            // ---- Engineering → % scaling ----
            IF enableScaling THEN
                pvPct := _ScaleToPct(pvEngFiltered,       pLoEng, pHiEng);
                spPct := _ScaleToPct(processSetpointAuto, pLoEng, pHiEng);
            ELSE
                pvPct := pvEngFiltered;        // already %
                spPct := processSetpointAuto;  // already %
            END_IF

            // ---- Manual path (HMI) ----
            manualCmd := LIMIT(0.0, processSetpointMan, 100.0);

            // Reverse/direct action by Kp sign
            IF reverseActing THEN
                kpUse := -ABS(kp);
            ELSE
                kpUse :=  ABS(kp);
            END_IF

            // ===================== PV HOLD behavior =====================
            // When PV hold active: keep motor energized, force reference=0.0,
            // and hold PID (avoid error/windup) by forcing SET=ACT and MAN=TRUE.
            IF pvHoldActive THEN

                deviceState := 'Running (PV hold: output inhibited)';
                vfdStartCmdOut := TRUE;        // keep energized
                running := TRUE;               // keep permissives (change to FALSE if you prefer)

                instPID(
                    ACT := pvPct,
                    SET := pvPct,              // hold: SET follows PV -> DIFF ~ 0
                    M_I := 0.0,                // forced output during hold
                    MAN := TRUE,               // hold PID
                    RST := resetPID,
                    KP  := kpUse,
                    TN  := tn,
                    TV  := tv,
                    LL  := outLowLimitPct,
                    LH  := outHighLimitPct,
                    Y   => yPID,
                    DIFF=> pidDiff,
                    LIM => pidLimited
                );

                // Output inhibited to zero, motor stays enabled
                controlOutputPct := 0.0;

            ELSE
                // ===================== Normal control =====================
                instPID(
                    ACT := pvPct,
                    SET := spPct,
                    M_I := manualCmd,
                    MAN := NOT autoMode,
                    RST := resetPID,
                    KP  := kpUse,
                    TN  := tn,
                    TV  := tv,
                    LL  := outLowLimitPct,
                    LH  := outHighLimitPct,
                    Y   => yPID,
                    DIFF=> pidDiff,
                    LIM => pidLimited
                );

                // Mode select, offset, clamp
                IF autoMode THEN
                    controlOutputPct := yPID;
                ELSE
                    controlOutputPct := manualCmd;
                END_IF

                controlOutputPct := LIMIT(outLowLimitPct, controlOutputPct + outputOffsetPct, outHighLimitPct);
            END_IF
        END_IF

    // ------------------------------------------------------------
    90: // Stopping (normal, de-energize)
        running := FALSE;
        controlOutputPct := 0.0;
        vfdStartCmdOut := FALSE;
        tonRunFbWait(IN := FALSE);

        // Return to Idle once stop released and safety OK
        IF NOT stopCommand AND allSafetyOK THEN
            deviceState := 'Idle';
            step := 0;
        END_IF

    // ------------------------------------------------------------
    ELSE
        running := FALSE;
        controlOutputPct := 0.0;
        deviceState := 'Idle';
        vfdStartCmdOut := FALSE;
        step := 0;
END_CASE;


// =============================== Status code ===============================
IF vfdFaultFeedback THEN
    statusCode := 2;             // Fault
ELSIF running THEN
    statusCode := 1;             // Running
ELSE
    statusCode := 0;             // Idle
END_IF

// HMI feedbacks & status (encapsulates PT1 displays and status code if desired)
_FeedbackDisplay();

// Setpoint input handling (encapsulates TUNE2-based HMI writes & nudges)
_SetpointInputControl();

METHOD _FeedbackDisplay
VAR_INPUT
END_VAR
//instPT1_WhiteWaterSiloDisplay
//whiteWaterLevelDisplay
// 5) HMI DISPLAY SIGNALS (filtered speeds/torques + GROUP status)
instPT1_SpeedDisplay(in := vfdEngFeedback, T := displayFilterTime, K := 1.0, out => vfdEngDisplay);
instPT1_TorqueDisplay (in := vfdTorqueFeedback , T := displayFilterTime, K := 1.0, out => vfdTorqueDisplay);
instPT1_ProcessFeedbackEngDisplay(in := wirePitLevel , T := displayFilterTime, K := 1.0, out => wirePitLevelDisplay);
instPT1_WhiteWaterSiloLevelDisplay(in := whiteWaterSiloLevel , T := displayFilterTime, K := 1.0, out => whiteWaterSiloLevelDisplay);
END_METHOD

// ============================ Helper ============================
METHOD PRIVATE _ScaleToPct : REAL
VAR_INPUT
    xEng  : REAL;  // value in engineering units
    loEng : REAL;  // min eng
    hiEng : REAL;  // max eng
END_VAR
VAR
    span : REAL;
    pct  : REAL;
END_VAR

span := hiEng - loEng;
IF span = 0.0 THEN
    _ScaleToPct := 0.0; // avoid div by zero
ELSE
    pct := (xEng - loEng) / span * 100.0;
    _ScaleToPct := LIMIT(0.0, pct, 100.0);
END_IF
END_METHOD

// ============================================================================
// METHOD: _SetpointInputControl
// Purpose: Handle HMI writes for manual output using OSCAT TUNE2. Any external
//          write to manualOutputPct bigger than the configured step will pulse
//          SET for one scan. No SU/SD buttons here (PressureCtrl doesn’t use them).
// Objetivo: Tratar escrita da HMI no manualOutputPct via TUNE2. Mudança externa
//           > passo gera pulso SET de 1 varredura. Sem botões ↑/↓ neste FB.
// ============================================================================
METHOD PRIVATE _SetpointInputControl
VAR
    spManClamped : REAL;
    spAutoClamped : REAL;
	
END_VAR
// Detect external write (> step): ignore tiny jitter
IF ABS(processSetpointMan - processSetpointManOld) > instTUNE2ManSetpoint.SS THEN
    // Clamp to output limits before writing (garante limites)
    spManClamped := LIMIT(outLowLimitPct, processSetpointMan, outHighLimitPct);

    // One-scan SET pulse into TUNE2 (pulso SET de 1 ciclo)
    instTUNE2ManSetpoint(
        SET_val := spManClamped,
        SET     := TRUE
    );
    instTUNE2ManSetpoint(SET := FALSE);

    // Remember applied value (memoriza)
    processSetpointManOld := processSetpointMan;
ELSE
    // Track last seen to avoid drift (rastreia último observado)
    processSetpointManOld := processSetpointMan;
END_IF;

// Keep TUNE2 active (no SU/SD in this FB)
instTUNE2ManSetpoint(
    SET      := FALSE,
    SU       := processSetpointManInc,
    SD       := processSetpointManDec,
    RST      := FALSE,
    SS       := 0.1,           // step reference (passo de referência)
    FS       := 0.0,                     // unused
    LIMIT_L  := outLowLimitPct,
    LIMIT_H  := outHighLimitPct,
    Y        => processSetpointMan
);




// Detect external write (> step): ignore tiny jitter
IF ABS(processSetpointAuto - processSetpointAutoOld) > instTUNE2AutoSetpoint.SS THEN
    // Clamp to output limits before writing (garante limites)
    spAutoClamped := LIMIT(0, processSetpointAuto, 100);

    // One-scan SET pulse into TUNE2 (pulso SET de 1 ciclo)
    instTUNE2AutoSetpoint(
        SET_val := spAutoClamped,
        SET     := TRUE
    );
    instTUNE2AutoSetpoint(SET := FALSE);

    // Remember applied value (memoriza)
    processSetpointAutoOld := processSetpointAuto;
ELSE
    // Track last seen to avoid drift (rastreia último observado)
    processSetpointAutoOld := processSetpointAuto;
END_IF;

// Keep TUNE2 active (no SU/SD in this FB)
instTUNE2AutoSetpoint(
    SET      := FALSE,
    SU       := processSetpointAutoInc,
    SD       := processSetpointAutoDec,
    RST      := FALSE,
    SS       := 0.1,           // step reference (passo de referência)
    FS       := 0.0,                     // unused
    LIMIT_L  := 0.0,
    LIMIT_H  := 100.0,
    Y        => processSetpointAuto
);
END_METHOD

END_FUNCTION_BLOCK

// ---- Function Blocks/PaperMachine/Auxiliary/FB_StockPumpFlowControl.TcPOU
(*
    FB_StockPumpFlowControl

    Purpose:
    Dedicated dry-stock flow controller for the Stock Pump (P1_100_UG05).
    The existing Mix Pump (P1_100_UG01) is the approach-flow fan/mix pump and
    is intentionally outside the scope of this function block.

    First delivery:
    Public interface and method declarations only. No control logic is active.
*)

FUNCTION_BLOCK FB_StockPumpFlowControl
VAR_INPUT
    // ===== General enable and sequence commands =====
    enable                              : BOOL;
    processPermissive                   : BOOL;
    startCommand                        : BOOL;
    stopCommand                         : BOOL;
    resetCommand                        : BOOL;
    autoMode                            : BOOL;   // TRUE=Automatic / FALSE=Manual
    machineRunning                      : BOOL;
    processStable                       : BOOL;

    // ===== Manual speed-reference adjustment =====
    stockPumpSetpointManInc             : BOOL;   // Increase manual speed reference
    stockPumpSetpointManDec             : BOOL;   // Decrease manual speed reference
    manualSetpointStepPct               : REAL := 0.1;

    // ===== Process inputs =====
    basisWeightSetpointGm2              : REAL;   // Desired basis weight [g/m2]
    effectiveWidthM                     : REAL;   // Effective sheet/jet width [m]
    wireSpeedMPM                        : REAL;   // Forming wire speed [m/min]
    stockConsistencyPct                 : REAL;   // Stock consistency [%], e.g. 3.5 = 3.5%
    stockConsistencySignalValid         : BOOL;
    refinedStockTankConsistencyPct      : REAL;   // Refined-stock tank consistency indication [%]
    refinedStockTankConsistencySignalValid : BOOL;
    stockFlowFeedbackM3h                : REAL;   // Measured suspension flow [m3/h]
    stockFlowSignalValid                : BOOL;
    stockTankLevelPct                   : REAL;   // Stock-tank level, already scaled [%]
    stockTankLevelSignalValid           : BOOL;

    // ===== Production correction factors =====
    recipeCalibrationFactor             : REAL := 1.0;
    operatorTrimFactor                  : REAL := 1.0;
    basisWeightLabGm2                   : REAL;
    calculateCalibrationCommand         : BOOL;

    // ===== PID parameters =====
    kp                                  : REAL := 1.0;
    tn                                  : REAL := 8.0;     // Integral time [s]
    tv                                  : REAL := 0.0;     // Derivative time [s]
    pidDeadbandM3h                      : REAL := 0.0;     // Flow deadband [m3/h]
    resetPID                            : BOOL;

    // ===== Process engineering limits =====
    stockDensityKgM3                    : REAL := 1000.0;
    minimumValidConsistencyPct          : REAL := 0.1;
    maximumValidConsistencyPct          : REAL := 10.0;
    minimumStockFlowM3h                 : REAL := 0.0;
    maximumStockFlowM3h                 : REAL := 250.0;
    standbyStockFlowM3h                 : REAL := 0.0;
    minimumAutomaticWireSpeedMPM        : REAL := 0.0;

    // ===== Calibration and trim limits =====
    minimumRecipeCalibrationFactor      : REAL := 0.5;
    maximumRecipeCalibrationFactor      : REAL := 1.5;
    minimumOperatorTrimFactor           : REAL := 0.95;
    maximumOperatorTrimFactor           : REAL := 1.05;

    // ===== Filters and ramps =====
    consistencyFilterTime               : TIME := T#5s;
    flowFeedbackFilterTime              : TIME := T#1s;
    stockTankLevelFilterTime            : TIME := T#2s;
    stockFlowSetpointRampUpM3hS         : REAL := 1.0;
    stockFlowSetpointRampDownM3hS       : REAL := 1.0;
    speedReferenceRampUpPctS            : REAL := 10.0;
    speedReferenceRampDownPctS          : REAL := 10.0;

    // ===== Speed-reference limits =====
    minimumSpeedReferencePct            : REAL := 0.0;
    maximumSpeedReferencePct            : REAL := 100.0;

    // ===== Signal fallback and alarm timing =====
    invalidConsistencyGraceTime         : TIME := T#5s;
    automaticStabilizationTime          : TIME := T#10s;
    flowDeviationWarningPct             : REAL := 5.0;
    flowDeviationAlarmPct               : REAL := 10.0;
    flowDeviationWarningDelay           : TIME := T#10s;
    flowDeviationAlarmDelay             : TIME := T#20s;

    // ===== Drive interface and supervision =====
    vfdReady                            : BOOL;
    vfdRunFeedback                      : BOOL;
    vfdFaultFeedback                    : BOOL;
    vfdRunFbTimeout                     : TIME := T#5s;
    vfdCurrentFeedback                  : REAL;
    vfdSpeedFeedbackPct                 : REAL;
    vfdTorqueFeedback                   : REAL;

    // ===== Safety and process interlocks =====
    safetyOk                            : BOOL := TRUE;
    estopOk                             : BOOL := TRUE;
    guardClosedOk                       : BOOL := TRUE;
    interlock1                          : BOOL := TRUE;
    interlock2                          : BOOL := TRUE;
    interlock3                          : BOOL := TRUE;
    interlock4                          : BOOL := TRUE;
    interlock5                          : BOOL := TRUE;
    interlock6                          : BOOL := TRUE;
END_VAR

VAR_IN_OUT
    // Existing HMI manual reference can be connected here without duplicating it.
    manualSpeedSetpointPct              : REAL;
END_VAR

VAR_OUTPUT
    // ===== Drive commands =====
    vfdStartCmdOut                      : BOOL;
    vfdResetCmdOut                      : BOOL;
    speedReferencePct                   : REAL;

    // ===== Flow and dry-mass calculation =====
    dryMassSetpointKgH                  : REAL;
    dryMassFeedbackKgH                  : REAL;
    stockFlowTheoreticalM3h             : REAL;
    stockFlowCorrectedM3h               : REAL;
    stockFlowLimitedM3h                 : REAL;
    stockFlowSetpointM3h                : REAL;
    stockFlowFeedbackFilteredM3h        : REAL;
    stockConsistencyFilteredPct         : REAL;
    stockConsistencyUsedPct             : REAL;

    // ===== Refined-stock tank consistency indication =====
    refinedStockTankConsistencyFilteredPct : REAL;
    refinedStockTankConsistencySignalInvalid : BOOL;

    // ===== Stock-tank indication =====
    stockTankLevelFilteredPct           : REAL;
    stockTankLevelSignalInvalid         : BOOL;

    // ===== PID diagnostics =====
    pidErrorM3h                         : REAL;
    pidOutputPct                        : REAL;
    pidOutputSaturated                  : BOOL;

    // ===== Calibration diagnostics =====
    suggestedCalibrationFactor         : REAL;
    suggestedCalibrationFactorValid    : BOOL;

    // ===== Validation and limitation status =====
    flowCalculationValid                : BOOL;
    automaticControlValid               : BOOL;
    automaticControlInvalid             : BOOL;
    consistencySignalInvalid            : BOOL;
    flowSignalInvalid                   : BOOL;
    basisWeightSetpointInvalid          : BOOL;
    effectiveWidthInvalid               : BOOL;
    wireSpeedInvalid                    : BOOL;
    calibrationFactorInvalid            : BOOL;
    operatorTrimFactorInvalid           : BOOL;
    flowSetpointLimited                 : BOOL;
    speedReferenceLimited              : BOOL;
    calculationUsingLastValidConsistency : BOOL;

    // ===== Deviation alarms =====
    flowDeviationWarning                : BOOL;
    flowDeviationAlarm                  : BOOL;
    warningActive                       : BOOL;
    alarmActive                         : BOOL;

    // ===== Operating state =====
    running                             : BOOL;
    controlActive                       : BOOL;
    manualActive                        : BOOL;
    automaticActive                     : BOOL;
    statusCode                          : INT;
    deviceState                         : STRING(80);

    // ===== Drive feedback displays =====
    vfdCurrentDisplay                   : REAL;
    vfdSpeedDisplayPct                  : REAL;
    vfdTorqueDisplay                    : REAL;
END_VAR

VAR
    // ===== Initialization and command edges =====
    firstScan                           : BOOL := TRUE;
    startCommandOld                     : BOOL;
    stopCommandOld                      : BOOL;
    resetCommandOld                     : BOOL;
    autoModeOld                         : BOOL;
    calculateCalibrationCommandOld      : BOOL;
    automaticControlValidOld            : BOOL;
    automaticActiveOld                  : BOOL;
    rStart                              : BOOL;
    rStop                               : BOOL;
    rReset                              : BOOL;
    rToAutomatic                        : BOOL;
    rToManual                           : BOOL;
    rCalculateCalibration               : BOOL;

    // ===== Drive sequence =====
    step                                : INT;
    runLatch                            : BOOL;
    allSafetyOk                         : BOOL;
    allInterlocksOk                     : BOOL;
    tonRunFeedbackWait                  : TON;

    // ===== Validity and fallback =====
    consistencyRawValid                 : BOOL;
    refinedStockTankConsistencyRawValid : BOOL;
    flowRawValid                        : BOOL;
    tankLevelRawValid                   : BOOL;
    consistencyAvailableForCalculation  : BOOL;
    engineeringConfigurationValid       : BOOL;
    lastValidConsistencyPct             : REAL;
    consistencyFilterInputPct           : REAL;
    refinedStockTankConsistencyFilterInputPct : REAL;
    flowFilterInputM3h                  : REAL;
    tankLevelFilterInputPct             : REAL;
    tonInvalidConsistency               : TON;

    // ===== Sanitized external limits =====
    consistencyLowUsePct                : REAL;
    consistencyHighUsePct               : REAL;
    flowLowUseM3h                       : REAL;
    flowHighUseM3h                      : REAL;
    speedLowUsePct                      : REAL;
    speedHighUsePct                     : REAL;
    calibrationLowUse                   : REAL;
    calibrationHighUse                  : REAL;
    operatorTrimLowUse                  : REAL;
    operatorTrimHighUse                 : REAL;

    // ===== Setpoint calculation and ramps =====
    stockFlowTargetBeforeLimitM3h       : REAL;
    suggestedCalibrationRaw             : REAL;
    speedReferenceTargetPct             : REAL;
    speedReferenceUnclampedPct          : REAL;
    manualCommandPct                    : REAL;
    manualSpeedSetpointOldPct           : REAL;
    manualSetpointStepUsePct            : REAL;
    manualSetpointInitialized           : BOOL;
    instManualSpeedSetpoint             : TUNE2;
    modeTransferHold                    : BOOL;
    instFlowSetpointRamp                : FB_Gen_SRamp;
    instSpeedReferenceRamp              : FB_Gen_SRamp;

    // ===== Filters and PID =====
    instConsistencyFilter               : FT_PT1;
    instRefinedStockTankConsistencyFilter : FT_PT1;
    instFlowFeedbackFilter              : FT_PT1;
    instStockTankLevelFilter            : FT_PT1;
    instPID                             : CTRL_PID;
    pidManualMode                       : BOOL;
    pidLimitedInternal                  : BOOL;

    // ===== Deviation supervision =====
    flowDeviationPct                    : REAL;
    deviationEvaluationEnabled          : BOOL;
    tonAutomaticStabilization           : TON;
    tonFlowDeviationWarning             : TON;
    tonFlowDeviationAlarm               : TON;
END_VAR

VAR CONSTANT
    cZeroTolerance                      : REAL := 0.000001;
    cRampVelocityLimit                  : REAL := 100000.0;
END_VAR

_Initialize();
_UpdateEdges();
_ValidateInputs();
_UpdateManualSetpoint();
_FilterProcessSignals();
_ManageConsistencyFallback();
_CalculateFlowSetpoint();
_RampFlowSetpoint();
_CalculateCalibrationSuggestion();
_HandleModeTransfer();
_RunDriveSequence();
_RunFlowController();
_RampSpeedReference();
_UpdateAlarmsAndDiagnostics();

// Calculate a suggested recipe factor without applying or persisting it.
METHOD PRIVATE _CalculateCalibrationSuggestion
IF rCalculateCalibration THEN
    suggestedCalibrationFactorValid := FALSE;

    IF processStable AND
       (basisWeightSetpointGm2 > cZeroTolerance) AND
       (basisWeightLabGm2 > cZeroTolerance) AND
       NOT calibrationFactorInvalid THEN

        suggestedCalibrationRaw := recipeCalibrationFactor *
                                  basisWeightSetpointGm2 /
                                  basisWeightLabGm2;

        suggestedCalibrationFactor := LIMIT(
            calibrationLowUse,
            suggestedCalibrationRaw,
            calibrationHighUse
        );

        suggestedCalibrationFactorValid :=
            (suggestedCalibrationRaw >= calibrationLowUse) AND
            (suggestedCalibrationRaw <= calibrationHighUse);
    END_IF;
END_IF;
END_METHOD

// Calculate dry mass and consistency-compensated stock-flow setpoint.
METHOD PRIVATE _CalculateFlowSetpoint
IF flowCalculationValid THEN
    // g/m2 * m * m/min * 0.06 = kg/h of dry stock.
    dryMassSetpointKgH := basisWeightSetpointGm2 * effectiveWidthM * wireSpeedMPM * 0.06;

    // kg/h / (kg/m3 * consistency fraction) = m3/h of stock suspension.
    IF (stockDensityKgM3 > cZeroTolerance) AND
       (stockConsistencyUsedPct > cZeroTolerance) THEN
        stockFlowTheoreticalM3h := dryMassSetpointKgH /
            (stockDensityKgM3 * stockConsistencyUsedPct * 0.01);
    ELSE
        stockFlowTheoreticalM3h := 0.0;
    END_IF;

    stockFlowCorrectedM3h := stockFlowTheoreticalM3h *
                             recipeCalibrationFactor *
                             operatorTrimFactor;

    IF wireSpeedMPM < MAX(0.0, minimumAutomaticWireSpeedMPM) THEN
        stockFlowTargetBeforeLimitM3h := standbyStockFlowM3h;
    ELSE
        stockFlowTargetBeforeLimitM3h := stockFlowCorrectedM3h;
    END_IF;

    stockFlowLimitedM3h := LIMIT(
        flowLowUseM3h,
        stockFlowTargetBeforeLimitM3h,
        flowHighUseM3h
    );

    flowSetpointLimited :=
        ABS(stockFlowLimitedM3h - stockFlowTargetBeforeLimitM3h) > cZeroTolerance;
ELSE
    dryMassSetpointKgH := 0.0;
    stockFlowTheoreticalM3h := 0.0;
    stockFlowCorrectedM3h := 0.0;
    stockFlowTargetBeforeLimitM3h := 0.0;
    stockFlowLimitedM3h := 0.0;
    flowSetpointLimited := FALSE;
END_IF;

IF consistencyAvailableForCalculation AND NOT flowSignalInvalid THEN
    dryMassFeedbackKgH := stockFlowFeedbackFilteredM3h *
                          stockDensityKgM3 *
                          stockConsistencyUsedPct * 0.01;
ELSE
    dryMassFeedbackKgH := 0.0;
END_IF;
END_METHOD

// Filter stock consistency, refined-stock indication, flow feedback and stock-tank level.
METHOD PRIVATE _FilterProcessSignals
// Invalid samples never enter the filters.
IF consistencyRawValid THEN
    consistencyFilterInputPct := stockConsistencyPct;
ELSIF lastValidConsistencyPct > cZeroTolerance THEN
    consistencyFilterInputPct := lastValidConsistencyPct;
ELSE
    consistencyFilterInputPct := consistencyLowUsePct;
END_IF;

instConsistencyFilter(
    in  := consistencyFilterInputPct,
    T   := consistencyFilterTime,
    K   := 1.0,
    out => stockConsistencyFilteredPct
);

// Indication-only: this measurement never participates in the flow calculation or PID.
IF refinedStockTankConsistencyRawValid THEN
    refinedStockTankConsistencyFilterInputPct := refinedStockTankConsistencyPct;
ELSE
    refinedStockTankConsistencyFilterInputPct := refinedStockTankConsistencyFilteredPct;
END_IF;

instRefinedStockTankConsistencyFilter(
    in  := refinedStockTankConsistencyFilterInputPct,
    T   := consistencyFilterTime,
    K   := 1.0,
    out => refinedStockTankConsistencyFilteredPct
);

IF flowRawValid THEN
    flowFilterInputM3h := stockFlowFeedbackM3h;
ELSE
    flowFilterInputM3h := stockFlowFeedbackFilteredM3h;
END_IF;

instFlowFeedbackFilter(
    in  := flowFilterInputM3h,
    T   := flowFeedbackFilterTime,
    K   := 1.0,
    out => stockFlowFeedbackFilteredM3h
);

// The tank level is indication-only and has no effect on pump control.
IF tankLevelRawValid THEN
    tankLevelFilterInputPct := stockTankLevelPct;
ELSE
    tankLevelFilterInputPct := stockTankLevelFilteredPct;
END_IF;

instStockTankLevelFilter(
    in  := tankLevelFilterInputPct,
    T   := stockTankLevelFilterTime,
    K   := 1.0,
    out => stockTankLevelFilteredPct
);
stockTankLevelFilteredPct := LIMIT(0.0, stockTankLevelFilteredPct, 100.0);

// Use the raw valid consistency while the PT1 output is still initializing.
IF consistencyRawValid THEN
    IF (stockConsistencyFilteredPct >= consistencyLowUsePct) AND
       (stockConsistencyFilteredPct <= consistencyHighUsePct) THEN
        stockConsistencyUsedPct := stockConsistencyFilteredPct;
    ELSE
        stockConsistencyUsedPct := stockConsistencyPct;
    END_IF;

    lastValidConsistencyPct := stockConsistencyUsedPct;
END_IF;
END_METHOD

// Prepare manual/automatic transitions for bumpless transfer.
METHOD PRIVATE _HandleModeTransfer
// Automatic to manual: initialize the manual reference with the active output.
IF rToManual THEN
    manualSpeedSetpointPct := LIMIT(speedLowUsePct, speedReferencePct, speedHighUsePct);
END_IF;

// Invalid automatic control falls back to a tracked manual reference.
IF autoMode AND automaticControlValidOld AND NOT automaticControlValid THEN
    manualSpeedSetpointPct := LIMIT(speedLowUsePct, speedReferencePct, speedHighUsePct);
END_IF;

// Track for one cycle before enabling automatic PID output.
IF rToAutomatic OR
   (autoMode AND automaticControlValid AND NOT automaticControlValidOld) THEN
    modeTransferHold := TRUE;
END_IF;

manualSpeedSetpointPct := LIMIT(
    speedLowUsePct,
    manualSpeedSetpointPct,
    speedHighUsePct
);
manualCommandPct := manualSpeedSetpointPct;

automaticControlValidOld := automaticControlValid;
END_METHOD

// Initialize internal states, retained values and safe output defaults.
METHOD PRIVATE _Initialize
IF firstScan THEN
    firstScan := FALSE;

    step := 0;
    runLatch := FALSE;
    speedReferencePct := 0.0;
    speedReferenceTargetPct := 0.0;
    stockFlowSetpointM3h := 0.0;

    startCommandOld := startCommand;
    stopCommandOld := stopCommand;
    resetCommandOld := resetCommand;
    autoModeOld := autoMode;
    calculateCalibrationCommandOld := calculateCalibrationCommand;
    automaticControlValidOld := FALSE;

    speedLowUsePct := LIMIT(0.0, MIN(minimumSpeedReferencePct, maximumSpeedReferencePct), 100.0);
    speedHighUsePct := LIMIT(speedLowUsePct, MAX(minimumSpeedReferencePct, maximumSpeedReferencePct), 100.0);
    manualSpeedSetpointPct := LIMIT(speedLowUsePct, manualSpeedSetpointPct, speedHighUsePct);

    IF stockConsistencySignalValid AND
       (stockConsistencyPct >= minimumValidConsistencyPct) AND
       (stockConsistencyPct <= maximumValidConsistencyPct) THEN
        lastValidConsistencyPct := stockConsistencyPct;
        stockConsistencyUsedPct := stockConsistencyPct;
    END_IF;
END_IF;
END_METHOD

// Hold the last valid consistency during the configured grace period.
METHOD PRIVATE _ManageConsistencyFallback
tonInvalidConsistency(
    IN := consistencySignalInvalid,
    PT := invalidConsistencyGraceTime
);

IF NOT consistencySignalInvalid THEN
    consistencyAvailableForCalculation := TRUE;
    calculationUsingLastValidConsistency := FALSE;

ELSIF (lastValidConsistencyPct > cZeroTolerance) AND NOT tonInvalidConsistency.Q THEN
    stockConsistencyUsedPct := lastValidConsistencyPct;
    consistencyAvailableForCalculation := TRUE;
    calculationUsingLastValidConsistency := TRUE;

ELSE
    consistencyAvailableForCalculation := FALSE;
    calculationUsingLastValidConsistency := FALSE;
END_IF;

flowCalculationValid :=
    engineeringConfigurationValid AND
    NOT basisWeightSetpointInvalid AND
    NOT effectiveWidthInvalid AND
    NOT wireSpeedInvalid AND
    NOT calibrationFactorInvalid AND
    NOT operatorTrimFactorInvalid AND
    consistencyAvailableForCalculation;

automaticControlValid :=
    enable AND
    processPermissive AND
    machineRunning AND
    flowCalculationValid AND
    NOT flowSignalInvalid AND
    vfdReady AND
    NOT vfdFaultFeedback AND
    allSafetyOk AND
    allInterlocksOk;

automaticControlInvalid := autoMode AND NOT automaticControlValid;
END_METHOD

// Apply the configured rate limits to the calculated stock-flow setpoint.
METHOD PRIVATE _RampFlowSetpoint
instFlowSetpointRamp(
    X          := stockFlowLimitedM3h,
    A_UP       := MAX(0.0, stockFlowSetpointRampUpM3hS),
    A_DN       := -MAX(0.0, stockFlowSetpointRampDownM3hS),
    VU_MAX     := cRampVelocityLimit,
    VD_MAX     := -cRampVelocityLimit,
    LIMIT_HIGH := flowHighUseM3h,
    LIMIT_LOW  := 0.0,
    RST        := NOT flowCalculationValid
);

IF flowCalculationValid THEN
    stockFlowSetpointM3h := LIMIT(
        0.0,
        instFlowSetpointRamp.Y,
        flowHighUseM3h
    );
ELSE
    stockFlowSetpointM3h := 0.0;
END_IF;
END_METHOD

// Apply the configured rate limits to the final drive-speed reference.
METHOD PRIVATE _RampSpeedReference
instSpeedReferenceRamp(
    X          := speedReferenceTargetPct,
    A_UP       := MAX(0.0, speedReferenceRampUpPctS),
    A_DN       := -MAX(0.0, speedReferenceRampDownPctS),
    VU_MAX     := cRampVelocityLimit,
    VD_MAX     := -cRampVelocityLimit,
    LIMIT_HIGH := speedHighUsePct,
    LIMIT_LOW  := 0.0,
    RST        := NOT running
);

IF running THEN
    speedReferencePct := LIMIT(
        0.0,
        instSpeedReferenceRamp.Y,
        speedHighUsePct
    );
ELSE
    speedReferencePct := 0.0;
END_IF;
END_METHOD

// Execute start, run, stop and drive-supervision state handling.
METHOD PRIVATE _RunDriveSequence
vfdStartCmdOut := FALSE;
vfdResetCmdOut := rReset;

// Immediate stop conditions.
IF stopCommand OR NOT enable OR NOT allSafetyOk OR vfdFaultFeedback THEN
    runLatch := FALSE;
    step := 90;
END_IF;

CASE step OF
    0: // Idle
        running := FALSE;
        vfdStartCmdOut := FALSE;
        deviceState := 'Idle';
        tonRunFeedbackWait(IN := FALSE);

        IF runLatch AND NOT stopCommand THEN
            IF NOT enable THEN
                deviceState := 'Start blocked: control disabled';
                runLatch := FALSE;
            ELSIF NOT allSafetyOk THEN
                deviceState := 'Start blocked: safety not OK';
                runLatch := FALSE;
            ELSIF NOT processPermissive OR NOT allInterlocksOk THEN
                deviceState := 'Start blocked: process interlock';
                runLatch := FALSE;
            ELSIF NOT vfdReady OR vfdFaultFeedback THEN
                deviceState := 'Start blocked: drive not ready';
                runLatch := FALSE;
            ELSE
                deviceState := 'Starting';
                vfdStartCmdOut := TRUE;
                step := 10;
            END_IF;
        END_IF;

    10: // Starting
        running := FALSE;
        vfdStartCmdOut := TRUE;
        deviceState := 'Starting: awaiting RUN feedback';
        tonRunFeedbackWait(IN := TRUE, PT := vfdRunFbTimeout);

        IF NOT enable OR stopCommand OR NOT allSafetyOk OR vfdFaultFeedback THEN
            runLatch := FALSE;
            step := 90;
        ELSIF NOT processPermissive OR NOT allInterlocksOk OR NOT vfdReady THEN
            runLatch := FALSE;
            step := 90;
        ELSIF vfdRunFeedback THEN
            tonRunFeedbackWait(IN := FALSE);
            step := 20;
        ELSIF tonRunFeedbackWait.Q THEN
            deviceState := 'Start failed: RUN feedback timeout';
            runLatch := FALSE;
            step := 90;
        END_IF;

    20: // Running
        running := TRUE;
        vfdStartCmdOut := TRUE;
        deviceState := 'Running';
        tonRunFeedbackWait(IN := FALSE);

        IF NOT enable OR stopCommand OR NOT allSafetyOk OR vfdFaultFeedback THEN
            runLatch := FALSE;
            step := 90;
        ELSIF NOT processPermissive OR NOT allInterlocksOk THEN
            runLatch := FALSE;
            step := 90;
        ELSIF NOT vfdReady OR NOT vfdRunFeedback THEN
            runLatch := FALSE;
            step := 90;
        ELSIF NOT runLatch THEN
            step := 90;
        END_IF;

    90: // Stopping
        running := FALSE;
        vfdStartCmdOut := FALSE;
        tonRunFeedbackWait(IN := FALSE);

        IF vfdFaultFeedback THEN
            deviceState := 'Fault from drive';
        ELSE
            deviceState := 'Stopping';
        END_IF;

        IF NOT stopCommand AND NOT vfdFaultFeedback AND allSafetyOk THEN
            step := 0;
        END_IF;

    ELSE
        running := FALSE;
        vfdStartCmdOut := FALSE;
        deviceState := 'Idle';
        runLatch := FALSE;
        step := 0;
END_CASE;
END_METHOD

// Execute the flow PID once per PLC cycle when control conditions are valid.
METHOD PRIVATE _RunFlowController
manualCommandPct := LIMIT(speedLowUsePct, manualSpeedSetpointPct, speedHighUsePct);

automaticActive := running AND autoMode AND automaticControlValid;
manualActive := running AND (NOT autoMode OR NOT automaticControlValid);
controlActive := automaticActive OR manualActive;

IF automaticActive AND NOT automaticActiveOld THEN
    modeTransferHold := TRUE;
END_IF;

// The PID is called exactly once per PLC cycle. In manual, stopped, invalid or
// transfer states, MAN/M_I tracks the active manual reference for anti-windup.
pidManualMode := NOT automaticActive OR modeTransferHold;

instPID(
    ACT  := stockFlowFeedbackFilteredM3h,
    SET  := stockFlowSetpointM3h,
    SUP  := MAX(0.0, pidDeadbandM3h),
    OFS  := 0.0,
    M_I  := manualCommandPct,
    MAN  := pidManualMode,
    RST  := resetPID OR NOT enable,
    KP   := ABS(kp),
    TN   := MAX(0.0, tn),
    TV   := MAX(0.0, tv),
    LL   := speedLowUsePct,
    LH   := speedHighUsePct,
    Y    => pidOutputPct,
    DIFF => pidErrorM3h,
    LIM  => pidLimitedInternal
);

pidOutputSaturated := pidLimitedInternal;

IF NOT running THEN
    speedReferenceUnclampedPct := 0.0;

ELSIF automaticActive AND NOT modeTransferHold THEN
    speedReferenceUnclampedPct := pidOutputPct;

ELSIF modeTransferHold THEN
    speedReferenceUnclampedPct := speedReferencePct;

ELSE
    // Explicit manual mode and invalid-automatic fallback both use this path.
    speedReferenceUnclampedPct := manualCommandPct;
END_IF;

IF running THEN
    speedReferenceTargetPct := LIMIT(
        speedLowUsePct,
        speedReferenceUnclampedPct,
        speedHighUsePct
    );

    speedReferenceLimited :=
        ABS(speedReferenceTargetPct - speedReferenceUnclampedPct) > cZeroTolerance;
ELSE
    speedReferenceTargetPct := 0.0;
    speedReferenceLimited := FALSE;
END_IF;

IF modeTransferHold THEN
    modeTransferHold := FALSE;
END_IF;

automaticActiveOld := automaticActive;
END_METHOD

// Evaluate flow deviation and consolidate status, warning and alarm outputs.
METHOD PRIVATE _UpdateAlarmsAndDiagnostics
tonAutomaticStabilization(
    IN := automaticActive,
    PT := automaticStabilizationTime
);

IF stockFlowSetpointM3h > cZeroTolerance THEN
    flowDeviationPct := ABS(stockFlowSetpointM3h - stockFlowFeedbackFilteredM3h) /
                        stockFlowSetpointM3h * 100.0;
ELSE
    flowDeviationPct := 0.0;
END_IF;

deviationEvaluationEnabled :=
    automaticActive AND
    vfdRunFeedback AND
    tonAutomaticStabilization.Q AND
    automaticControlValid AND
    (stockFlowSetpointM3h > cZeroTolerance);

tonFlowDeviationWarning(
    IN := deviationEvaluationEnabled AND
          (flowDeviationPct >= MAX(0.0, flowDeviationWarningPct)),
    PT := flowDeviationWarningDelay
);

tonFlowDeviationAlarm(
    IN := deviationEvaluationEnabled AND
          (flowDeviationPct >= MAX(0.0, flowDeviationAlarmPct)),
    PT := flowDeviationAlarmDelay
);

flowDeviationWarning := tonFlowDeviationWarning.Q;
flowDeviationAlarm := tonFlowDeviationAlarm.Q;

warningActive :=
    flowDeviationWarning OR
    calculationUsingLastValidConsistency OR
    flowSetpointLimited OR
    speedReferenceLimited;

alarmActive :=
    flowDeviationAlarm OR
    vfdFaultFeedback OR
    (running AND automaticControlInvalid);

IF vfdFaultFeedback THEN
    statusCode := 2;
ELSIF running THEN
    statusCode := 1;
ELSE
    statusCode := 0;
END_IF;

vfdCurrentDisplay := vfdCurrentFeedback;
vfdSpeedDisplayPct := vfdSpeedFeedbackPct;
vfdTorqueDisplay := vfdTorqueFeedback;
END_METHOD

// Detect command and mode-transition edges.
METHOD PRIVATE _UpdateEdges
rStart := startCommand AND NOT startCommandOld;
rStop := stopCommand AND NOT stopCommandOld;
rReset := resetCommand AND NOT resetCommandOld;
rToAutomatic := autoMode AND NOT autoModeOld;
rToManual := NOT autoMode AND autoModeOld;
rCalculateCalibration := calculateCalibrationCommand AND NOT calculateCalibrationCommandOld;

startCommandOld := startCommand;
stopCommandOld := stopCommand;
resetCommandOld := resetCommand;
autoModeOld := autoMode;
calculateCalibrationCommandOld := calculateCalibrationCommand;

IF rStart THEN
    runLatch := TRUE;
END_IF;

IF rStop OR stopCommand THEN
    runLatch := FALSE;
END_IF;
END_METHOD

// Apply the existing HMI increase/decrease commands to the manual speed reference.
METHOD PRIVATE _UpdateManualSetpoint
manualSetpointStepUsePct := MAX(cZeroTolerance, ABS(manualSetpointStepPct));

// Synchronize the tuner after an HMI numeric entry or an internal bumpless transfer.
IF NOT manualSetpointInitialized OR
   (ABS(manualSpeedSetpointPct - manualSpeedSetpointOldPct) > cZeroTolerance) THEN
    instManualSpeedSetpoint(
        SET_val := LIMIT(speedLowUsePct, manualSpeedSetpointPct, speedHighUsePct),
        SET     := TRUE
    );
    instManualSpeedSetpoint(SET := FALSE);
    manualSetpointInitialized := TRUE;
END_IF;

// Preserve the established HMI button behavior. Opposite commands cancel each other.
instManualSpeedSetpoint(
    SET     := FALSE,
    SU      := stockPumpSetpointManInc AND NOT stockPumpSetpointManDec,
    SD      := stockPumpSetpointManDec AND NOT stockPumpSetpointManInc,
    RST     := FALSE,
    SS      := manualSetpointStepUsePct,
    FS      := 0.0,
    LIMIT_L := speedLowUsePct,
    LIMIT_H := speedHighUsePct,
    Y       => manualSpeedSetpointPct
);

manualSpeedSetpointPct := LIMIT(
    speedLowUsePct,
    manualSpeedSetpointPct,
    speedHighUsePct
);
manualSpeedSetpointOldPct := manualSpeedSetpointPct;
END_METHOD

// Validate process signals, configuration limits and correction factors.
METHOD PRIVATE _ValidateInputs
// Sanitize all configurable ranges before they are used by LIMIT or the PID.
consistencyLowUsePct := MAX(cZeroTolerance, MIN(minimumValidConsistencyPct, maximumValidConsistencyPct));
consistencyHighUsePct := MAX(consistencyLowUsePct, MAX(minimumValidConsistencyPct, maximumValidConsistencyPct));

flowLowUseM3h := MAX(0.0, MIN(minimumStockFlowM3h, maximumStockFlowM3h));
flowHighUseM3h := MAX(flowLowUseM3h, MAX(minimumStockFlowM3h, maximumStockFlowM3h));

speedLowUsePct := LIMIT(0.0, MIN(minimumSpeedReferencePct, maximumSpeedReferencePct), 100.0);
speedHighUsePct := LIMIT(speedLowUsePct, MAX(minimumSpeedReferencePct, maximumSpeedReferencePct), 100.0);

calibrationLowUse := MAX(cZeroTolerance, MIN(minimumRecipeCalibrationFactor, maximumRecipeCalibrationFactor));
calibrationHighUse := MAX(calibrationLowUse, MAX(minimumRecipeCalibrationFactor, maximumRecipeCalibrationFactor));

operatorTrimLowUse := MAX(cZeroTolerance, MIN(minimumOperatorTrimFactor, maximumOperatorTrimFactor));
operatorTrimHighUse := MAX(operatorTrimLowUse, MAX(minimumOperatorTrimFactor, maximumOperatorTrimFactor));

consistencyRawValid := stockConsistencySignalValid AND
                       (stockConsistencyPct >= consistencyLowUsePct) AND
                       (stockConsistencyPct <= consistencyHighUsePct);
refinedStockTankConsistencyRawValid := refinedStockTankConsistencySignalValid AND
                                       (refinedStockTankConsistencyPct >= consistencyLowUsePct) AND
                                       (refinedStockTankConsistencyPct <= consistencyHighUsePct);

flowRawValid := stockFlowSignalValid AND (stockFlowFeedbackM3h >= 0.0);
tankLevelRawValid := stockTankLevelSignalValid AND
                     (stockTankLevelPct >= 0.0) AND
                     (stockTankLevelPct <= 100.0);

consistencySignalInvalid := NOT consistencyRawValid;
refinedStockTankConsistencySignalInvalid := NOT refinedStockTankConsistencyRawValid;
flowSignalInvalid := NOT flowRawValid;
stockTankLevelSignalInvalid := NOT tankLevelRawValid;
basisWeightSetpointInvalid := basisWeightSetpointGm2 <= 0.0;
effectiveWidthInvalid := effectiveWidthM <= 0.0;
wireSpeedInvalid := wireSpeedMPM < 0.0;

calibrationFactorInvalid :=
    (minimumRecipeCalibrationFactor <= 0.0) OR
    (maximumRecipeCalibrationFactor < minimumRecipeCalibrationFactor) OR
    (recipeCalibrationFactor < calibrationLowUse) OR
    (recipeCalibrationFactor > calibrationHighUse);

operatorTrimFactorInvalid :=
    (minimumOperatorTrimFactor <= 0.0) OR
    (maximumOperatorTrimFactor < minimumOperatorTrimFactor) OR
    (operatorTrimFactor < operatorTrimLowUse) OR
    (operatorTrimFactor > operatorTrimHighUse);

engineeringConfigurationValid :=
    (stockDensityKgM3 > cZeroTolerance) AND
    (minimumValidConsistencyPct > 0.0) AND
    (maximumValidConsistencyPct >= minimumValidConsistencyPct) AND
    (minimumStockFlowM3h >= 0.0) AND
    (maximumStockFlowM3h >= minimumStockFlowM3h) AND
    (minimumSpeedReferencePct >= 0.0) AND
    (maximumSpeedReferencePct <= 100.0) AND
    (maximumSpeedReferencePct >= minimumSpeedReferencePct);

allSafetyOk := safetyOk AND estopOk AND guardClosedOk;
allInterlocksOk := interlock1 AND interlock2 AND interlock3 AND
                   interlock4 AND interlock5 AND interlock6;

// Final consolidated validity is updated after consistency fallback handling.
flowCalculationValid := FALSE;
automaticControlValid := FALSE;
automaticControlInvalid := autoMode;
END_METHOD

END_FUNCTION_BLOCK

// ---- Function Blocks/PaperMachine/Auxiliary/FB_ConsistencyControllerModbusTcp.TcPOU
FUNCTION_BLOCK FB_ConsistencyControllerModbusTcp
VAR_INPUT PERSISTENT
    deviceConfig : ST_ConsistencyControllerConfig;
END_VAR

VAR_OUTPUT
    controllerInputs : ST_ConsistencyControllerInputs;
END_VAR

VAR
    fbReadRegisters : FB_MBReadRegs;
    fbDelay         : TON;
    aRegisters     : ARRAY[0..5] OF WORD;
    dwProcessValue : DWORD;
    eState         : USINT;
    bExecute       : BOOL;
    bDelayEnable   : BOOL;
    tActiveDelay   : TIME;
    nIndex         : INT;
END_VAR

VAR CONSTANT
    STATE_DISABLED       : USINT := 0;
    STATE_STARTUP_DELAY  : USINT := 10;
    STATE_POLL_DELAY     : USINT := 20;
    STATE_WAIT_RESPONSE  : USINT := 30;
    EXPECTED_BYTE_COUNT  : UDINT := 12;
    ERROR_INVALID_LENGTH : UDINT := 16#E0010001;
END_VAR

// SEGURANCA DE COMISSIONAMENTO:
// Este FB implementa somente leitura Modbus FC03 por meio de FB_MBReadRegs.
// Nao existem blocos FB_MBWrite* nem chamadas FC05/FC06/FC15/FC16 nesta implementacao.
// Com deviceConfig.bEnable=FALSE, nenhuma requisicao TCP e disparada para o equipamento.
// Qualquer escrita futura exige revisao, validacao em bancada e um intertravamento dedicado.

// Uma unica requisicao FC03 le o bloco continuo 4001..4006.
// O bloco e instanciado uma vez por equipamento pelo metodo do MAIN.
controllerInputs.bEnabled := deviceConfig.bEnable;
controllerInputs.bBusy := fbReadRegisters.bBusy;
bExecute := FALSE;

// O mesmo TON atende a defasagem de partida e o periodo entre leituras.
bDelayEnable := (eState = STATE_STARTUP_DELAY) OR (eState = STATE_POLL_DELAY);
IF eState = STATE_STARTUP_DELAY THEN
    tActiveDelay := deviceConfig.tStartupDelay;
ELSE
    tActiveDelay := deviceConfig.tPollInterval;
END_IF

fbDelay(
    IN := bDelayEnable,
    PT := tActiveDelay
);

CASE eState OF
    STATE_DISABLED:
        controllerInputs.bOnline := FALSE;
        IF deviceConfig.bEnable THEN
            eState := STATE_STARTUP_DELAY;
        END_IF

    STATE_STARTUP_DELAY,
    STATE_POLL_DELAY:
        IF NOT deviceConfig.bEnable THEN
            eState := STATE_DISABLED;
        ELSIF fbDelay.Q THEN
            bExecute := TRUE;
            eState := STATE_WAIT_RESPONSE;
        END_IF

    STATE_WAIT_RESPONSE:
        // A primeira passagem por este estado ocorre depois da borda de Execute.
        // Ao terminar, Busy cai e os dados/diagnosticos ja estao estaveis.
        IF NOT fbReadRegisters.bBusy THEN
            controllerInputs.cbLastRead := fbReadRegisters.cbRead;

            IF fbReadRegisters.bError OR (fbReadRegisters.cbRead <> EXPECTED_BYTE_COUNT) THEN
                controllerInputs.bOnline := FALSE;
                controllerInputs.udiFailedReads := controllerInputs.udiFailedReads + 1;
                controllerInputs.udiConsecutiveErrors := controllerInputs.udiConsecutiveErrors + 1;

                IF fbReadRegisters.bError THEN
                    controllerInputs.nErrorId := fbReadRegisters.nErrId;
                ELSE
                    controllerInputs.nErrorId := ERROR_INVALID_LENGTH;
                END_IF
            ELSE
                FOR nIndex := 0 TO 5 DO
                    controllerInputs.aRawRegisters[nIndex] := aRegisters[nIndex];
                END_FOR

                controllerInputs.nSetpointRaw := WORD_TO_INT(aRegisters[0]);

                // PV e um DINT distribuido nos registros 4002 e 4003.
                // A ordem de words pode ser invertida na configuracao sem alterar o FB.
                IF deviceConfig.bPvLowWordFirst THEN
                    dwProcessValue := SHL(WORD_TO_DWORD(aRegisters[2]), 16)
                                      OR WORD_TO_DWORD(aRegisters[1]);
                ELSE
                    dwProcessValue := SHL(WORD_TO_DWORD(aRegisters[1]), 16)
                                      OR WORD_TO_DWORD(aRegisters[2]);
                END_IF

                controllerInputs.diProcessValueRaw := DWORD_TO_DINT(dwProcessValue);
                controllerInputs.nManipulatedValueRaw := WORD_TO_INT(aRegisters[3]);
                controllerInputs.nCalibrationRaw := WORD_TO_INT(aRegisters[4]);
                controllerInputs.nModeRaw := WORD_TO_INT(aRegisters[5]);

                controllerInputs.rSetpoint := INT_TO_REAL(controllerInputs.nSetpointRaw) / 100.0;
                controllerInputs.rProcessValue := DINT_TO_REAL(controllerInputs.diProcessValueRaw) / 100.0;
                controllerInputs.rManipulatedValuePct := INT_TO_REAL(controllerInputs.nManipulatedValueRaw) / 10.0;
                controllerInputs.nCalibration := controllerInputs.nCalibrationRaw;
                controllerInputs.bCalibrationValid := (controllerInputs.nCalibrationRaw >= 1)
                                                      AND (controllerInputs.nCalibrationRaw <= 3);
                controllerInputs.bAutomatic := controllerInputs.nModeRaw = 1;
                controllerInputs.bModeValid := (controllerInputs.nModeRaw = 0)
                                               OR (controllerInputs.nModeRaw = 1);

                controllerInputs.bOnline := TRUE;
                controllerInputs.nErrorId := 0;
                controllerInputs.udiSuccessfulReads := controllerInputs.udiSuccessfulReads + 1;
                controllerInputs.udiConsecutiveErrors := 0;
                controllerInputs.uliLastSuccessFileTime := F_GetSystemTime();
            END_IF

            IF deviceConfig.bEnable THEN
                eState := STATE_POLL_DELAY;
            ELSE
                eState := STATE_DISABLED;
            END_IF
        END_IF

ELSE
    eState := STATE_DISABLED;
END_CASE

// O FB Beckhoff deve ser chamado em todos os ciclos, inclusive durante Busy.
fbReadRegisters(
    sIPAddr := deviceConfig.sIpAddress,
    nTCPPort := deviceConfig.uiTcpPort,
    nUnitID := deviceConfig.byUnitId,
    nQuantity := 6,
    nMBAddr := deviceConfig.uiFirstRegister,
    cbLength := SIZEOF(aRegisters),
    pDestAddr := ADR(aRegisters),
    bExecute := bExecute,
    tTimeout := deviceConfig.tResponseTimeout
);

// Atualiza Busy novamente para refletir a chamada realizada neste ciclo.
controllerInputs.bBusy := fbReadRegisters.bBusy;

END_FUNCTION_BLOCK

// ---- Function Blocks/DELTA - MS300/FB_DELTA_C2000_ETC.TcPOU
FUNCTION_BLOCK FB_DELTA_C2000_ETC



//======================================================================
// Persistent Configuration Inputs
//======================================================================
VAR_INPUT PERSISTENT
	
    deviceConfig            : C2000_DEV_CONFIG;       // Device-specific configuration (scaling, limits, etc.)

END_VAR

//======================================================================
// Runtime Inputs
//======================================================================
VAR_INPUT
	
    speedSetpoint           : REAL;                		// Motor speed reference to be written to drive
	torqueSetpoint			: REAL;						// Torque limit if running as torque
    commandWord             : C2000_CONTROLWORD;      	// Control word to drive (start, stop, etc.)
    digitalOutputs          : C2000_DIGITAL_OUTPUTS;  	// Digital output values to send to drive
    analogOutputs           : C2000_ANALOG_OUTPUTS;   	// Analog output values to send to drive
	
END_VAR

//======================================================================
// Runtime Outputs
//======================================================================
VAR_OUTPUT
	
    statusWord              : C2000_STATUSWORD;       // Current status word read from drive
    digitalInputs           : C2000_DIGITAL_INPUTS;   // Current status of digital inputs from drive
    analogInputs            : C2000_ANALOG_INPUTS;    // Current status of analog inputs from drive
    motorSpeedRPM             : REAL;                   // Actual motor speed read from drive in RPM
    motorSpeedEng             : REAL;                   // Actual motor speed read from drive in enginering units scaled
    outputCurrent           : REAL;                   // Output current read from drive
    outputTorque            : REAL;                   // Output torque read from drive
    currentErrorCode        : UINT;                   // Current C2000 Plus error code (CiA 402 object 603Fh)
    faultCodeAtTrip         : UINT;                   // Error code latched when the fault is detected
    faultTorqueAtTrip       : REAL;                   // Scaled output torque latched with the fault
    faultEventCounter       : UDINT;                  // Increments for each new fault/code while faulted
	
	
	pdoSpeedSet			: INT;
	
	
END_VAR

//======================================================================
// Internal Variables
//======================================================================
VAR
    PDOS                    : C2000_PDOS;             // Process Data Object structure containing drive mappings
    // One-shot + pulse for fault reset
    rTrigReset : R_TRIG;
    tReset     : TOF;
	
    // Base OMS bits default (keep your logic)
    b0_swOn, b1_enVolt, b2_qStopOK, b3_enOp : BOOL;
    b4, b5, b6, b7_faultReset, b8_halt      : BOOL;
    cw                                       : WORD;

    // Reset sequencer helpers
 //   rTrigReset        : R_TRIG;   // detect rising edge of reset command
    tResetClear       : TON;      // phase 1: clear all bits (control word = 0)
    tResetPulse       : TON;      // phase 2: pulse bit7 = 1
    resetSeqActive    : BOOL;     // TRUE while running either phase
    resetClearPt      : TIME := T#500MS;    // adjust if your drive needs longer clear
    resetPulsePt      : TIME := T#1000ms;  // 1 second fault-reset pulse	
    faultWasActive    : BOOL;     // Previous-cycle state used by the diagnostic latch

END_VAR

(*==============================================================================================================================
CPNTeck - Automação Industrial
(c)Copyright 2025 All Rights Reserved
_______________________________________________________________________________________________________________________________
Library: N/A
Tested with: CX920
Engineering: TwinCAT 3
Restrictions: -
Requirements: N/A
Functionality: This function block communicates with a Delta MS300 drive over Modbus RTU. It reads process values such as
               motor speed, current, torque, status words, digital and analog inputs, and writes control commands and 
               setpoints to the drive. The block includes timeout monitoring and state-based communication handling.
Support: fabio@cpnteck.com.br
Note: Parameter comments are only available in language 'English (United States)'

_______________________________________________________________________________________________________________________________
Change log table:

Version         | Date         | Expert in charge   | Changes applied
01.00.01        | 31.05.2025   | Fabio Campion      | Initial implementation for MS300 drive Modbus RTU communication
==============================================================================================================================*)

_StatusWord();       // Method to handle the status word of the drive
_DigitalInputs();    // Method to process the status of digital inputs
_AnalogInputs();     // Method to handle analog input values

_CommandWord();      // Method to set or process the command word for the drive
_DigitalOutputs();   // Method to manage the status of digital outputs
_AnalogOutputs();    // Method to handle analog output values
_SetOperationMode();
_FeedBackVariables(); // Method to process feedback variables from the drive
_FaultSnapshot();     // Latch code and torque at the instant of a drive fault
_SpeedReference();         // Method to set or process the setpoint values
_TorqueReference();

METHOD PRIVATE _AnalogInputs
VAR_INPUT
END_VAR
END_METHOD

METHOD PRIVATE _AnalogOutputs
VAR_INPUT
END_VAR
END_METHOD

METHOD PRIVATE _CommandWord
VAR_INPUT
END_VAR
(*
VAR
    // Internal
    b0_swOn, b1_enVolt, b2_qStopOK, b3_enOp, b4, b5, b6 : BOOL;
    b7_faultReset, b8_halt                              : BOOL;
    cw                                                  : UINT;
END_VAR
*)

b4 := 1;
b5 := 1;
b6 := 1;


// ---------- 1) Base state from commands (bits 0..3) ----------
IF commandWord.quickStop THEN
    // Quick-stop has highest priority: keep voltage/switch-on, clear enable op, force bit2=0
    b0_swOn    := TRUE;
    b1_enVolt  := TRUE;
    b2_qStopOK := FALSE;  // bit2=0 => quick stop active
    b3_enOp    := FALSE;

ELSIF commandWord.enableDrive THEN
    // Enable Operation: 1,1,1,1
    b0_swOn    := TRUE;
    b1_enVolt  := TRUE;
    b2_qStopOK := TRUE;
    b3_enOp    := TRUE;

ELSIF commandWord.stopRequest THEN
    // Switch On (ready but not enabled): 1,1,1,0
    b0_swOn    := TRUE;
    b1_enVolt  := TRUE;
    b2_qStopOK := TRUE;
    b3_enOp    := FALSE;

ELSE
    // Shutdown (safe, DC bus on): 0,1,1,0
    b0_swOn    := FALSE;
    b1_enVolt  := TRUE;
    b2_qStopOK := TRUE;
    b3_enOp    := FALSE;
END_IF


// ---------- 2) Halt (bit8) ----------
b8_halt := commandWord.halt;

// ---------- 3) Fault Reset as 1000 ms pulse (bit7) ----------
rTrigReset(CLK := commandWord.faultResetCmd);
tReset(IN := rTrigReset.Q, PT := T#1000ms);
b7_faultReset := tReset.Q;

// ---------- 4) Pack bits into 16-bit control word ----------
cw := 0; // bits 9..15 remain 0 unless you set them later

// base (0..3)
IF b0_swOn    THEN cw := cw OR 16#0001; END_IF; // bit0
IF b1_enVolt  THEN cw := cw OR 16#0002; END_IF; // bit1
IF b2_qStopOK THEN cw := cw OR 16#0004; END_IF; // bit2
IF b3_enOp    THEN cw := cw OR 16#0008; END_IF; // bit3

// OMS (4..6) — use correct masks
IF b4          THEN cw := cw OR 16#0010; END_IF; // bit4
IF b5          THEN cw := cw OR 16#0020; END_IF; // bit5
IF b6          THEN cw := cw OR 16#0040; END_IF; // bit6

// bit7 (fault reset pulse) and bit8 (halt)
IF b7_faultReset THEN cw := cw OR 16#0080; END_IF; // bit7
IF b8_halt       THEN cw := cw OR 16#0100; END_IF; // bit8

// Bits 9..15 reserved = 0
PDOS.PlcToDrv.controlWord := cw;



//==============================================================
// CIA402 CONTROL WORD BUILD — with proper reset sequence
//==============================================================
(*

//==============================================================
// 0) Edge-detect RESET command and run the two-phase sequence
//==============================================================
rTrigReset(CLK := commandWord.faultResetCmd);

// Start sequence on rising edge
IF rTrigReset.Q THEN
    resetSeqActive := TRUE;
    // (Re)start clear phase
    tResetClear(IN := TRUE, PT := resetClearPt);
    // ensure pulse is off until clear finishes
    tResetPulse(IN := FALSE, PT := resetPulsePt);
END_IF;

// Advance/reset timers when sequence is active
IF resetSeqActive THEN
    // Phase 1: CLEAR (control word = 0)
    tResetClear(IN := tResetClear.IN, PT := resetClearPt);

    // When clear finishes, start pulse (only once)
    IF tResetClear.Q AND NOT tResetPulse.IN THEN
        tResetClear(IN := FALSE, PT := resetClearPt);     // stop clear timer
        tResetPulse(IN := TRUE,  PT := resetPulsePt);     // start pulse
    END_IF;

    // Run pulse
    tResetPulse(IN := tResetPulse.IN, PT := resetPulsePt);

    // Sequence ends when pulse finishes
    IF tResetPulse.Q THEN
        tResetPulse(IN := FALSE, PT := resetPulsePt);
        resetSeqActive := FALSE;
    END_IF;
END_IF;


//==============================================================
// 1) NORMAL PACKING (only used when NOT resetting)
//==============================================================

// Default OMS high (per your original)
b4 := TRUE;  // bit4 mask 0x0010
b5 := TRUE;  // bit5 mask 0x0020
b6 := TRUE;  // bit6 mask 0x0040

// ---------- 1) Base state from commands (bits 0..3) ----------
IF commandWord.quickStop THEN
    // Quick-stop has highest priority
    b0_swOn    := TRUE;
    b1_enVolt  := TRUE;
    b2_qStopOK := FALSE; // quick stop active
    b3_enOp    := FALSE;

ELSIF commandWord.enableDrive THEN
    // Enable Operation: 1,1,1,1
    b0_swOn    := TRUE;
    b1_enVolt  := TRUE;
    b2_qStopOK := TRUE;
    b3_enOp    := TRUE;

ELSIF commandWord.stopRequest THEN
    // Switch On (ready but not enabled): 1,1,1,0
    b0_swOn    := TRUE;
    b1_enVolt  := TRUE;
    b2_qStopOK := TRUE;
    b3_enOp    := FALSE;

ELSE
    // Shutdown (safe, DC bus on): 0,1,1,0
    b0_swOn    := FALSE;
    b1_enVolt  := TRUE;
    b2_qStopOK := TRUE;
    b3_enOp    := FALSE;
END_IF;

// ---------- 2) Halt (bit8) ----------
b8_halt := commandWord.halt;


//==============================================================
// 2) BUILD CONTROL WORD — with RESET SEQUENCE OVERRIDE
//==============================================================
cw := 0;

// If reset sequence is active, override everything
IF resetSeqActive THEN
    // Phase 1: CLEAR → send 0x0000
    IF NOT tResetClear.Q THEN
//        cw := 16#0000;
        cw := 16#0080;
		

    // Phase 2: PULSE → send only bit7 = 1 (0x0080)
    ELSIF tResetClear.Q AND NOT tResetPulse.Q THEN
//        cw := 16#0080;
        cw := 16#0000;
		
    END_IF;

ELSE
    // Normal packing
    // base (0..3)
    IF b0_swOn    THEN cw := cw OR 16#0001; END_IF; // bit0
    IF b1_enVolt  THEN cw := cw OR 16#0002; END_IF; // bit1
    IF b2_qStopOK THEN cw := cw OR 16#0004; END_IF; // bit2
    IF b3_enOp    THEN cw := cw OR 16#0008; END_IF; // bit3

    // OMS (4..6)
    IF b4          THEN cw := cw OR 16#0010; END_IF; // bit4
    IF b5          THEN cw := cw OR 16#0020; END_IF; // bit5
    IF b6          THEN cw := cw OR 16#0040; END_IF; // bit6

    // bit7 (fault reset) — now driven EXCLUSIVELY by the sequencer, so keep low here
    // b7_faultReset := FALSE;

    // bit8 (halt)
    IF b8_halt       THEN cw := cw OR 16#0100; END_IF; // bit8

    // Bits 9..15 remain 0 unless set elsewhere
END_IF;

// Push to PDO
PDOS.PlcToDrv.controlWord := cw;
*)
END_METHOD

METHOD PRIVATE _DigitalInputs 
VAR_INPUT
END_VAR
END_METHOD

METHOD PRIVATE _DigitalOutputs : BOOL
VAR_INPUT
END_VAR
END_METHOD

METHOD PRIVATE _FaultSnapshot
VAR_INPUT
END_VAR
currentErrorCode := PDOS.DrvToPLC.errorCode;

// Capture the first fault cycle and any subsequent error-code change while
// the drive remains faulted. The values stay latched after a drive reset so
// the historian cannot lose a short-lived diagnostic between ADS polls.
IF statusWord.fault AND
   ((NOT faultWasActive) OR (currentErrorCode <> faultCodeAtTrip)) THEN
    faultCodeAtTrip := currentErrorCode;
    faultTorqueAtTrip := outputTorque;
    faultEventCounter := faultEventCounter + 1;
END_IF;

faultWasActive := statusWord.fault;
END_METHOD

METHOD PRIVATE _FeedBackVariables
VAR_INPUT
END_VAR

VAR
	
	OutputTorqueAux : REAL;

END_VAR
// Calculate the actual motor speed
motorSpeedRPM := DINT_TO_REAL(PDOS.DrvToPLC.velocityActualValue);
// Calculate the actual motor speed in meters per minute
motorSpeedEng := _Scale(
    X := DINT_TO_REAL(PDOS.DrvToPLC.velocityActualValue), 
    I_LO := deviceConfig.MotorSpeedInputLow, 
    I_HI := deviceConfig.MotorSpeedInputHigh, 
    O_LO := deviceConfig.MotorSpeedMPMOutputLow, 
    O_HI := deviceConfig.MotorSpeedMPMOutputHigh
);

// Calculate the actual output torque
OutputTorque := _Scale(
    X := INT_TO_REAL(PDOS.DrvToPLC.torqueActualValue), 
    I_LO := deviceConfig.OutputTorqueInputLow, 
    I_HI := deviceConfig.OutputTorqueInputHigh, 
    O_LO := deviceConfig.OutputTorqueOutputLow, 
    O_HI := deviceConfig.OutputTorqueOutputHigh
);
END_METHOD

METHOD PRIVATE _Scale : REAL
VAR_INPUT
	
	X : REAL;
	I_LO : REAL;
	I_HI : REAL;
	O_LO : REAL;
	O_HI : REAL;
	
END_VAR
IF I_LO = I_HI THEN
	_Scale := O_LO;
ELSE
	_Scale := (O_HI - O_LO) / (I_HI - I_LO) * (LIMIT(I_LO, X, I_HI) - I_LO) + O_LO;
END_IF;
END_METHOD

METHOD PRIVATE _SetOperationMode
VAR_INPUT
END_VAR
CASE deviceConfig.operationMode OF

    E_C2000_ModeOfOperation.Reserved_0:
        PDOS.PlcToDrv.modesOfOperation := 0;
        ; // Reserved - no action

    E_C2000_ModeOfOperation.ProfilePositionMode:
        PDOS.PlcToDrv.modesOfOperation := 1;
        ; // Profile Position Mode handling

    E_C2000_ModeOfOperation.VelocityMode:
        PDOS.PlcToDrv.modesOfOperation := 2;
        ; // Velocity Mode handling

    E_C2000_ModeOfOperation.Reserved_3:
        PDOS.PlcToDrv.modesOfOperation := 3;
        ; // Reserved - no action

    E_C2000_ModeOfOperation.ProfileTorqueMode:
        PDOS.PlcToDrv.modesOfOperation := 4;
		
        ; // Profile Torque Mode handling

    E_C2000_ModeOfOperation.Reserved_5:
        PDOS.PlcToDrv.modesOfOperation := 5;
        ; // Reserved - no action

    E_C2000_ModeOfOperation.HomingMode:
        PDOS.PlcToDrv.modesOfOperation := 6;
        ; // Homing Mode handling

    E_C2000_ModeOfOperation.Reserved_7:
        PDOS.PlcToDrv.modesOfOperation := 7;
        ; // Reserved - no action

    E_C2000_ModeOfOperation.CyclicSynchronousPositionMode:
        PDOS.PlcToDrv.modesOfOperation := 8;
        ; // Cyclic Synchronous Position Mode handling

    E_C2000_ModeOfOperation.Reserved_9:
        PDOS.PlcToDrv.modesOfOperation := 9;
        ; // Reserved - no action

    E_C2000_ModeOfOperation.CyclicSynchronousTorqueMode:
        PDOS.PlcToDrv.modesOfOperation := 10;
        ; // Cyclic Synchronous Torque Mode handling

ELSE
    PDOS.PlcToDrv.modesOfOperation := 2;
    ; // Fallback: Undefined mode, default to reserved

END_CASE
END_METHOD

METHOD PRIVATE _SpeedReference
VAR_INPUT
END_VAR
// --- Update Velocity Target Setpoint (signed INT) ---
PDOS.PlcToDrv.vlTargetVelocity := REAL_TO_INT(_Scale(
    X    := speedSetpoint, 
    I_LO := deviceConfig.speedSetpointInputLow, 
    I_HI := deviceConfig.speedSetpointInputHigh, 
    O_LO := deviceConfig.speedSetpointOutputLow, 
    O_HI := deviceConfig.speedSetpointOutputHigh));

	PDOS.PlcToDrv.maxMotorSpeed := PDOS.PlcToDrv.vlTargetVelocity;
	
	pdoSpeedSet := PDOS.PlcToDrv.vlTargetVelocity;
END_METHOD

METHOD PRIVATE _StatusWord
VAR_INPUT
END_VAR
// --- Map raw statusword bits to structured fields ---------------------------
StatusWord.readyToSwitchOn     := PDOS.DrvToPLC.StatusWord.0;   // Bit 0
StatusWord.switchedOn          := PDOS.DrvToPLC.StatusWord.1;   // Bit 1
StatusWord.operationEnabled    := PDOS.DrvToPLC.StatusWord.2;   // Bit 2
StatusWord.fault               := PDOS.DrvToPLC.StatusWord.3;   // Bit 3
StatusWord.voltageEnabled      := PDOS.DrvToPLC.StatusWord.4;   // Bit 4
StatusWord.quickStop           := PDOS.DrvToPLC.StatusWord.5;   // Bit 5
StatusWord.switchOnDisabled    := PDOS.DrvToPLC.StatusWord.6;   // Bit 6
StatusWord.warning             := PDOS.DrvToPLC.StatusWord.7;   // Bit 7
StatusWord.reserved1           := PDOS.DrvToPLC.StatusWord.8;   // Bit 8 (reserved)
StatusWord.remote              := PDOS.DrvToPLC.StatusWord.9;   // Bit 9
StatusWord.targetReached       := PDOS.DrvToPLC.StatusWord.10;  // Bit 10
StatusWord.internalLimitActive := PDOS.DrvToPLC.StatusWord.11;  // Bit 11
END_METHOD

METHOD PRIVATE _TorqueReference
VAR_INPUT
END_VAR

VAR
END_VAR


IF deviceConfig.torqueLimiterEnabled THEN
	
	// --- Update Velocity Target Setpoint (signed INT) ---
	PDOS.PlcToDrv.maxTorque := REAL_TO_UINT(_Scale(
		X    := torqueSetpoint, 
		I_LO := deviceConfig.torqueSetpointInputLow, 
		I_HI := deviceConfig.torqueSetpointInputHigh, 
		O_LO := deviceConfig.torqueSetpointOutputLow, 
		O_HI := deviceConfig.torqueSetpointOutputHigh) + deviceConfig.torqueDif);
		
ELSE
	
	PDOS.PlcToDrv.maxTorque := REAL_TO_UINT (deviceConfig.torqueSetpointOutputHigh);
	
END_IF
END_METHOD

END_FUNCTION_BLOCK

// ---- Function Blocks/IOs/Beckhoff/EL3052 - Ai 2 x 4-20MA - 12bit/FB_EL3052.TcPOU
FUNCTION_BLOCK FB_EL3052
VAR_INPUT PERSISTENT

	deviceConfig    : EL3052_DEV_CONFIG; // Configuration settings for the CT121F device
	
END_VAR
VAR_OUTPUT
		
	Channel1  : REAL;
	Channel2  : REAL;
	
END_VAR
VAR
	    PDOS : EL3052_PDOS; // Process Data Objects for RWPT01D communication
END_VAR


_AnalogInputs();

METHOD PRIVATE _AnalogInputs
VAR_INPUT
END_VAR
// Calculate the actual motor speed
Channel1 := _Scale(
    X := DINT_TO_REAL(PDOS.HwToPLC.Channel1.Value), 
    I_LO := deviceConfig.channel1InputLow, 
    I_HI := deviceConfig.channel1InputHigh, 
    O_LO := deviceConfig.channel1OutputLow, 
    O_HI := deviceConfig.channel1OutputHigh
);

// Calculate the actual motor speed
Channel2 := _Scale(
    X := DINT_TO_REAL(PDOS.HwToPLC.Channel2.Value), 
    I_LO := deviceConfig.channe12InputLow, 
    I_HI := deviceConfig.channe12InputHigh, 
    O_LO := deviceConfig.channe12OutputLow, 
    O_HI := deviceConfig.channe12OutputHigh
);
END_METHOD

METHOD PRIVATE _Scale : REAL
VAR_INPUT
	
	X : REAL;
	I_LO : REAL;
	I_HI : REAL;
	O_LO : REAL;
	O_HI : REAL;
	
END_VAR
IF I_LO = I_HI THEN
	_Scale := O_LO;
ELSE
	_Scale := (O_HI - O_LO) / (I_HI - I_LO) * (LIMIT(I_LO, X, I_HI) - I_LO) + O_LO;
END_IF;
END_METHOD

END_FUNCTION_BLOCK

// ---- Function Blocks/IOs/Beckhoff/EL4024 - AQ 4 x 4-20MA/FB_EL4024.TcPOU
FUNCTION_BLOCK FB_EL4024
VAR_INPUT PERSISTENT

	deviceConfig    : EL4024_DEV_CONFIG; // Configuration settings for the CT121F device
	
END_VAR
VAR_INPUT
		
	Channel1  : REAL;
	Channel2  : REAL;
	Channel3  : REAL;
	Channel4  : REAL;
	
END_VAR
VAR
	    PDOS : EL4024_PDOS; // Process Data Objects for RWPT01D communication
END_VAR

_AnalogOutputs();

METHOD PRIVATE _AnalogOutputs
VAR_INPUT
END_VAR
// Calculate the actual motor speed
PDOS.HwToPLC.Channel1 := REAL_TO_INT(_Scale(
    X	 := Channel1, 
    I_LO := deviceConfig.channel1InputLow, 
    I_HI := deviceConfig.channel1InputHigh, 
    O_LO := deviceConfig.channel1OutputLow, 
    O_HI := deviceConfig.channel1OutputHigh
));
// Calculate the actual motor speed
PDOS.HwToPLC.Channel2 := REAL_TO_INT(_Scale(
    X	 := Channel2, 
    I_LO := deviceConfig.channel2InputLow, 
    I_HI := deviceConfig.channel2InputHigh, 
    O_LO := deviceConfig.channel2OutputLow, 
    O_HI := deviceConfig.channel2OutputHigh
));
// Calculate the actual motor speed
PDOS.HwToPLC.Channel3 := REAL_TO_INT(_Scale(
    X	 := Channel3, 
    I_LO := deviceConfig.channel3InputLow, 
    I_HI := deviceConfig.channel3InputHigh, 
    O_LO := deviceConfig.channel3OutputLow, 
    O_HI := deviceConfig.channel3OutputHigh
));
// Calculate the actual motor speed
PDOS.HwToPLC.Channel4 := REAL_TO_INT(_Scale(
    X	 := Channel4, 
    I_LO := deviceConfig.channel4InputLow, 
    I_HI := deviceConfig.channel4InputHigh, 
    O_LO := deviceConfig.channel4OutputLow, 
    O_HI := deviceConfig.channel4OutputHigh
));
END_METHOD

METHOD PRIVATE _Scale : REAL
VAR_INPUT
	
	X : REAL;
	I_LO : REAL;
	I_HI : REAL;
	O_LO : REAL;
	O_HI : REAL;
	
END_VAR
IF I_LO = I_HI THEN
	_Scale := O_LO;
ELSE
	_Scale := (O_HI - O_LO) / (I_HI - I_LO) * (LIMIT(I_LO, X, I_HI) - I_LO) + O_LO;
END_IF;
END_METHOD

END_FUNCTION_BLOCK

// ---- Function Blocks/IOs/Beckhoff/EL6910 - TwinSAFE PLC/FB_EL6910.TcPOU
FUNCTION_BLOCK FB_EL6910
VAR_INPUT
	
		errorAcknowledgement : BOOL;
		run  : BOOL;
		safetyReset : BOOL;

END_VAR
VAR_OUTPUT

	eStop1Status	: EL6910_ESTOP_STATUS;
	eStop1Diagnostics : EL6910_ESTOP_DIGNOSTICS;

	eStop2Status	: EL6910_ESTOP_STATUS;
	eStop2Diagnostics : EL6910_ESTOP_DIGNOSTICS;

	eStop3Status	: EL6910_ESTOP_STATUS;
	eStop3Diagnostics : EL6910_ESTOP_DIGNOSTICS;

	eStop4Status	: EL6910_ESTOP_STATUS;
	eStop4Diagnostics : EL6910_ESTOP_DIGNOSTICS;
	

END_VAR
VAR
	    PDOS : EL6910_PDOS; // Process Data Objects for EL6910 communication
		EStop1DiagOld: INT;
		EStop2DiagOld: INT;
		EStop3DiagOld: INT;
		EStop4DiagOld: INT;

		
		
END_VAR


_eStopDiagnostics();
_eStopStatus();
_SafetyPLC();

METHOD PRIVATE _eStopDiagnostics
VAR_INPUT
END_VAR
//==============================================================
// E-STOP 1
//==============================================================

eStop1Diagnostics.discrepancyErrGroup1       := PDOS.HwToPLC.EStop1Diag.0;
eStop1Diagnostics.discrepancyErrGroup2       := PDOS.HwToPLC.EStop1Diag.1;
eStop1Diagnostics.discrepancyErrGroup3       := PDOS.HwToPLC.EStop1Diag.2;
eStop1Diagnostics.discrepancyErrGroup4       := PDOS.HwToPLC.EStop1Diag.3;

eStop1Diagnostics.edmMonitoringErr1          := PDOS.HwToPLC.EStop1Diag.4;
eStop1Diagnostics.edmMonitoringErr2          := PDOS.HwToPLC.EStop1Diag.5;

// Bits 6 and 7 are skipped (not used)

eStop1Diagnostics.discrepancyErrGroup1_Safe  := PDOS.HwToPLC.EStop1Diag.8;
eStop1Diagnostics.discrepancyErrGroup2_Safe  := PDOS.HwToPLC.EStop1Diag.9;
eStop1Diagnostics.discrepancyErrGroup3_Safe  := PDOS.HwToPLC.EStop1Diag.10;
eStop1Diagnostics.discrepancyErrGroup4_Safe  := PDOS.HwToPLC.EStop1Diag.11;


//==============================================================
// E-STOP 2
//==============================================================
eStop2Diagnostics.discrepancyErrGroup1       := PDOS.HwToPLC.EStop2Diag.0;
eStop2Diagnostics.discrepancyErrGroup2       := PDOS.HwToPLC.EStop2Diag.1;
eStop2Diagnostics.discrepancyErrGroup3       := PDOS.HwToPLC.EStop2Diag.2;
eStop2Diagnostics.discrepancyErrGroup4       := PDOS.HwToPLC.EStop2Diag.3;

eStop2Diagnostics.edmMonitoringErr1          := PDOS.HwToPLC.EStop2Diag.4;
eStop2Diagnostics.edmMonitoringErr2          := PDOS.HwToPLC.EStop2Diag.5;

// Bits 6 and 7 skipped (not used)

eStop2Diagnostics.discrepancyErrGroup1_Safe  := PDOS.HwToPLC.EStop2Diag.8;
eStop2Diagnostics.discrepancyErrGroup2_Safe  := PDOS.HwToPLC.EStop2Diag.9;
eStop2Diagnostics.discrepancyErrGroup3_Safe  := PDOS.HwToPLC.EStop2Diag.10;
eStop2Diagnostics.discrepancyErrGroup4_Safe  := PDOS.HwToPLC.EStop2Diag.11;


//==============================================================
// E-STOP 3
//==============================================================
eStop3Diagnostics.discrepancyErrGroup1       := PDOS.HwToPLC.EStop3Diag.0;
eStop3Diagnostics.discrepancyErrGroup2       := PDOS.HwToPLC.EStop3Diag.1;
eStop3Diagnostics.discrepancyErrGroup3       := PDOS.HwToPLC.EStop3Diag.2;
eStop3Diagnostics.discrepancyErrGroup4       := PDOS.HwToPLC.EStop3Diag.3;

eStop3Diagnostics.edmMonitoringErr1          := PDOS.HwToPLC.EStop3Diag.4;
eStop3Diagnostics.edmMonitoringErr2          := PDOS.HwToPLC.EStop3Diag.5;

// Bits 6 and 7 skipped (not used)

eStop3Diagnostics.discrepancyErrGroup1_Safe  := PDOS.HwToPLC.EStop3Diag.8;
eStop3Diagnostics.discrepancyErrGroup2_Safe  := PDOS.HwToPLC.EStop3Diag.9;
eStop3Diagnostics.discrepancyErrGroup3_Safe  := PDOS.HwToPLC.EStop3Diag.10;
eStop3Diagnostics.discrepancyErrGroup4_Safe  := PDOS.HwToPLC.EStop3Diag.11;


//==============================================================
// E-STOP 4
//==============================================================
eStop4Diagnostics.discrepancyErrGroup1       := PDOS.HwToPLC.EStop4Diag.0;
eStop4Diagnostics.discrepancyErrGroup2       := PDOS.HwToPLC.EStop4Diag.1;
eStop4Diagnostics.discrepancyErrGroup3       := PDOS.HwToPLC.EStop4Diag.2;
eStop4Diagnostics.discrepancyErrGroup4       := PDOS.HwToPLC.EStop4Diag.3;

eStop4Diagnostics.edmMonitoringErr1          := PDOS.HwToPLC.EStop4Diag.4;
eStop4Diagnostics.edmMonitoringErr2          := PDOS.HwToPLC.EStop4Diag.5;

// Bits 6 and 7 skipped (not used)

eStop4Diagnostics.discrepancyErrGroup1_Safe  := PDOS.HwToPLC.EStop4Diag.8;
eStop4Diagnostics.discrepancyErrGroup2_Safe  := PDOS.HwToPLC.EStop4Diag.9;
eStop4Diagnostics.discrepancyErrGroup3_Safe  := PDOS.HwToPLC.EStop4Diag.10;
eStop4Diagnostics.discrepancyErrGroup4_Safe  := PDOS.HwToPLC.EStop4Diag.11;
END_METHOD

METHOD PRIVATE _eStopStatus
VAR_INPUT
END_VAR


IF PDOS.HwToPLC.EStop1State <> EStop1DiagOld THEN
	
	// Reset all states to FALSE
	eStop1Status.estopState_RUN        := FALSE;
	eStop1Status.estopState_STOP       := FALSE;
	eStop1Status.estopState_SAFE       := FALSE;
	eStop1Status.estopState_ERROR      := FALSE;
	eStop1Status.estopState_RESET      := FALSE;
	eStop1Status.estopState_START      := FALSE;
	eStop1Status.estopState_DELAYOUT   := FALSE;

	CASE PDOS.HwToPLC.EStop1State OF
		
		1: eStop1Status.estopState_RUN        := TRUE;
		2: eStop1Status.estopState_STOP       := TRUE;
		3: eStop1Status.estopState_SAFE       := TRUE;
		4: eStop1Status.estopState_ERROR      := TRUE;
		5: eStop1Status.estopState_RESET      := TRUE;
		6: eStop1Status.estopState_START      := TRUE;
		8: eStop1Status.estopState_DELAYOUT   := TRUE;
	
	END_CASE
END_IF
	
EStop1DiagOld := PDOS.HwToPLC.EStop1State;


//==============================================================
// E-STOP 2
//==============================================================
IF PDOS.HwToPLC.EStop2State <> EStop2DiagOld THEN

    // Reset all states to FALSE
    eStop2Status.estopState_RUN       := FALSE;
    eStop2Status.estopState_STOP      := FALSE;
    eStop2Status.estopState_SAFE      := FALSE;
    eStop2Status.estopState_ERROR     := FALSE;
    eStop2Status.estopState_RESET     := FALSE;
    eStop2Status.estopState_START     := FALSE;
    eStop2Status.estopState_DELAYOUT  := FALSE;

    CASE PDOS.HwToPLC.EStop2State OF
        1: eStop2Status.estopState_RUN      := TRUE;
        2: eStop2Status.estopState_STOP     := TRUE;
        3: eStop2Status.estopState_SAFE     := TRUE;
        4: eStop2Status.estopState_ERROR    := TRUE;
        5: eStop2Status.estopState_RESET    := TRUE;
        6: eStop2Status.estopState_START    := TRUE;
        8: eStop2Status.estopState_DELAYOUT := TRUE;
    END_CASE
END_IF;

EStop2DiagOld := PDOS.HwToPLC.EStop2State;


//==============================================================
// E-STOP 3
//==============================================================
IF PDOS.HwToPLC.EStop3State <> EStop3DiagOld THEN

    // Reset all states to FALSE
    eStop3Status.estopState_RUN       := FALSE;
    eStop3Status.estopState_STOP      := FALSE;
    eStop3Status.estopState_SAFE      := FALSE;
    eStop3Status.estopState_ERROR     := FALSE;
    eStop3Status.estopState_RESET     := FALSE;
    eStop3Status.estopState_START     := FALSE;
    eStop3Status.estopState_DELAYOUT  := FALSE;

    CASE PDOS.HwToPLC.EStop3State OF
        1: eStop3Status.estopState_RUN      := TRUE;
        2: eStop3Status.estopState_STOP     := TRUE;
        3: eStop3Status.estopState_SAFE     := TRUE;
        4: eStop3Status.estopState_ERROR    := TRUE;
        5: eStop3Status.estopState_RESET    := TRUE;
        6: eStop3Status.estopState_START    := TRUE;
        8: eStop3Status.estopState_DELAYOUT := TRUE;
    END_CASE
END_IF;

EStop3DiagOld := PDOS.HwToPLC.EStop3State;


//==============================================================
// E-STOP 4
//==============================================================
IF PDOS.HwToPLC.EStop4State <> EStop4DiagOld THEN

    // Reset all states to FALSE
    eStop4Status.estopState_RUN       := FALSE;
    eStop4Status.estopState_STOP      := FALSE;
    eStop4Status.estopState_SAFE      := FALSE;
    eStop4Status.estopState_ERROR     := FALSE;
    eStop4Status.estopState_RESET     := FALSE;
    eStop4Status.estopState_START     := FALSE;
    eStop4Status.estopState_DELAYOUT  := FALSE;

    CASE PDOS.HwToPLC.EStop4State OF
        1: eStop4Status.estopState_RUN      := TRUE;
        2: eStop4Status.estopState_STOP     := TRUE;
        3: eStop4Status.estopState_SAFE     := TRUE;
        4: eStop4Status.estopState_ERROR    := TRUE;
        5: eStop4Status.estopState_RESET    := TRUE;
        6: eStop4Status.estopState_START    := TRUE;
        8: eStop4Status.estopState_DELAYOUT := TRUE;
    END_CASE
END_IF;

EStop4DiagOld := PDOS.HwToPLC.EStop4State;
END_METHOD

METHOD PRIVATE _SafetyPLC
VAR_INPUT
END_VAR

PDOS.PlcToHw.Run := run;
PDOS.PlcToHw.safetyReset := safetyReset;

PDOS.PlcToHw.ErrorAcknowledgement := errorAcknowledgement;
END_METHOD

END_FUNCTION_BLOCK

// ---- Function Blocks/IOs/Beckhoff/EL4004 - AQ 4 x 0-10V/FB_EL4004.TcPOU
FUNCTION_BLOCK FB_EL4004
VAR_INPUT PERSISTENT

	deviceConfig    : EL4004_DEV_CONFIG; // Configuration settings for the CT121F device
	
END_VAR
VAR_INPUT
		
	Channel1  : REAL;
	Channel2  : REAL;
	Channel3  : REAL;
	Channel4  : REAL;
	
END_VAR
VAR
	    PDOS : EL4004_PDOS; // Process Data Objects for RWPT01D communication
END_VAR

_AnalogOutputs();

METHOD PRIVATE _AnalogOutputs
VAR_INPUT
END_VAR
// Calculate the actual motor speed
PDOS.HwToPLC.Channel1 := REAL_TO_INT(_Scale(
    X	 := Channel1, 
    I_LO := deviceConfig.channel1InputLow, 
    I_HI := deviceConfig.channel1InputHigh, 
    O_LO := deviceConfig.channel1OutputLow, 
    O_HI := deviceConfig.channel1OutputHigh
));
// Calculate the actual motor speed
PDOS.HwToPLC.Channel2 := REAL_TO_INT(_Scale(
    X	 := Channel2, 
    I_LO := deviceConfig.channel2InputLow, 
    I_HI := deviceConfig.channel2InputHigh, 
    O_LO := deviceConfig.channel2OutputLow, 
    O_HI := deviceConfig.channel2OutputHigh
));
// Calculate the actual motor speed
PDOS.HwToPLC.Channel3 := REAL_TO_INT(_Scale(
    X	 := Channel3, 
    I_LO := deviceConfig.channel3InputLow, 
    I_HI := deviceConfig.channel3InputHigh, 
    O_LO := deviceConfig.channel3OutputLow, 
    O_HI := deviceConfig.channel3OutputHigh
));
// Calculate the actual motor speed
PDOS.HwToPLC.Channel4 := REAL_TO_INT(_Scale(
    X	 := Channel4, 
    I_LO := deviceConfig.channel4InputLow, 
    I_HI := deviceConfig.channel4InputHigh, 
    O_LO := deviceConfig.channel4OutputLow, 
    O_HI := deviceConfig.channel4OutputHigh
));
END_METHOD

METHOD PRIVATE _Scale : REAL
VAR_INPUT
	
	X : REAL;
	I_LO : REAL;
	I_HI : REAL;
	O_LO : REAL;
	O_HI : REAL;
	
END_VAR
IF I_LO = I_HI THEN
	_Scale := O_LO;
ELSE
	_Scale := (O_HI - O_LO) / (I_HI - I_LO) * (LIMIT(I_LO, X, I_HI) - I_LO) + O_LO;
END_IF;
END_METHOD

END_FUNCTION_BLOCK

// ---- Function Blocks/IOs/Beckhoff/EL3154 - Ai 4 x 4-20MA - 16bit/FB_EL3154.TcPOU
FUNCTION_BLOCK FB_EL3154
VAR_INPUT PERSISTENT

	deviceConfig    : EL3154_DEV_CONFIG; // Configuration settings for the CT121F device
	
END_VAR
VAR_OUTPUT
		
	Channel1  : REAL;
	Channel2  : REAL;
	Channel3  : REAL;
	Channel4  : REAL;

END_VAR
VAR
	    PDOS : EL3154_PDOS; // Process Data Objects for RWPT01D communication
END_VAR


_AnalogInputs();

METHOD PRIVATE _AnalogInputs
VAR_INPUT
END_VAR
// Calculate the actual motor speed
Channel1 := _Scale(
    X := DINT_TO_REAL(PDOS.HwToPLC.Channel1.Value), 
    I_LO := deviceConfig.channel1InputLow, 
    I_HI := deviceConfig.channel1InputHigh, 
    O_LO := deviceConfig.channel1OutputLow, 
    O_HI := deviceConfig.channel1OutputHigh
);

// Calculate the actual motor speed
Channel2 := _Scale(
    X := DINT_TO_REAL(PDOS.HwToPLC.Channel2.Value), 
    I_LO := deviceConfig.channe12InputLow, 
    I_HI := deviceConfig.channe12InputHigh, 
    O_LO := deviceConfig.channe12OutputLow, 
    O_HI := deviceConfig.channe12OutputHigh
);

// Calculate the actual motor speed
Channel3 := _Scale(
    X := DINT_TO_REAL(PDOS.HwToPLC.Channel3.Value), 
    I_LO := deviceConfig.channel3InputLow, 
    I_HI := deviceConfig.channel3InputHigh, 
    O_LO := deviceConfig.channel3OutputLow, 
    O_HI := deviceConfig.channel3OutputHigh
);

// Calculate the actual motor speed
Channel4 := _Scale(
    X := DINT_TO_REAL(PDOS.HwToPLC.Channel4.Value), 
    I_LO := deviceConfig.channel4InputLow, 
    I_HI := deviceConfig.channel4InputHigh, 
    O_LO := deviceConfig.channel4OutputLow, 
    O_HI := deviceConfig.channel4OutputHigh
);
END_METHOD

METHOD PRIVATE _Scale : REAL
VAR_INPUT
	
	X : REAL;
	I_LO : REAL;
	I_HI : REAL;
	O_LO : REAL;
	O_HI : REAL;
	
END_VAR
IF I_LO = I_HI THEN
	_Scale := O_LO;
ELSE
	_Scale := (O_HI - O_LO) / (I_HI - I_LO) * (LIMIT(I_LO, X, I_HI) - I_LO) + O_LO;
END_IF;
END_METHOD

END_FUNCTION_BLOCK

// ---- Function Blocks/PaperMachine/Auxiliary/FB_SoftstarterSimple.TcPOU
(*
  FUNCTION_BLOCK FB_SoftstarterSimple
  Purpose:
    - Simplified softstarter sequencing with only Start/Stop.
    - No line/bypass contactor or overlap timing.
  Behavior:
    - Start when: startCommand=TRUE, softstarter OK, and all interlocks OK.
    - Optional: current proof (disabled by default).
    - Stop is immediate and safe (de-energize START).
  Notes:
    - Interface aligned with previous style for easy migration.
*)

FUNCTION_BLOCK FB_SoftstarterSimple
VAR_INPUT
    // Commands & interlocks
    startCommand         : BOOL;      // Start command
    stopCommand          : BOOL;      // Stop command
    sofstarterOK         : BOOL;      // Softstarter healthy/ready

    interlock1           : BOOL := TRUE; // External interlock 1
    interlock2           : BOOL := TRUE; // External interlock 2
    interlock3           : BOOL := TRUE; // External interlock 3
    interlock4           : BOOL := TRUE; // External interlock 4

    // Optional current proof (disabled if currentProofEnabled=FALSE)
    currentProofEnabled  : BOOL := FALSE;
    motorCurrentFeedback : REAL;      // Measured motor current
    minCurrentThreshold  : REAL := 30.0;    // Threshold for proof
    currentProofTime     : TIME := T#20S;   // Time above threshold
END_VAR

VAR_OUTPUT
    faultActive          : BOOL;      // Latched fault (clears when Start/Stop released)
    running              : BOOL;      // TRUE while RUNNING
    softstarterStart     : BOOL;      // START signal to softstarter
    deviceState          : STRING(80);// Human-readable state
END_VAR

VAR
    // State & edges
    step                 : INT;       // 0=IDLE, 10=STARTING, 20=PROVING, 30=RUN
    startCommandOld      : BOOL;
    rStart               : BOOL;

    // Timers
    tonCurrentProof      : TON;

    // Helpers
    allInterlocksOK      : BOOL;
END_VAR

// ============================ Edges, interlocks, defaults ============================
rStart := startCommand AND NOT startCommandOld;
startCommandOld := startCommand;

allInterlocksOK := interlock1 AND interlock2 AND interlock3 AND interlock4;

// Default state text
deviceState := 'Idle';

// Clear latched fault when both commands are released
IF NOT startCommand AND NOT stopCommand THEN
    faultActive := FALSE;
END_IF

// Immediate safe stop
IF stopCommand THEN
    softstarterStart := FALSE;
    running          := FALSE;
    tonCurrentProof(IN := FALSE);
    step := 0;
    deviceState := 'Stopped';
END_IF

// If a fault is active, hold safe idle
IF faultActive THEN
    softstarterStart := FALSE;
    running          := FALSE;
    tonCurrentProof(IN := FALSE);
    step := 0;
END_IF


// ================================= State machine ===================================
IF startCommand AND NOT stopCommand AND NOT faultActive THEN

    // Check preconditions (only at/into sequence)
    IF (NOT sofstarterOK) OR (NOT allInterlocksOK) THEN
        faultActive := TRUE;
        deviceState := 'Fault: interlock/softstarter not OK';
        softstarterStart := FALSE;
        running := FALSE;
        tonCurrentProof(IN := FALSE);
        step := 0;

    ELSE
        CASE step OF
            0:  // IDLE -> STARTING
                deviceState      := 'Starting';
                softstarterStart := TRUE;      // Command softstarter to start
                running          := FALSE;

                // Reset current proof
                tonCurrentProof(IN := FALSE);
                step := 10;

            10: // STARTING -> either PROVING or RUN (if proof disabled)
                deviceState := 'Starting';
                IF currentProofEnabled AND (currentProofTime > T#0s) THEN
                    step := 20;
                ELSE
                    // No proof required -> go straight to RUN
                    step := 30;
                END_IF

            20: // PROVING current above threshold
                deviceState := 'Proving current';
                IF ABS(motorCurrentFeedback) >= minCurrentThreshold THEN
                    tonCurrentProof(IN := TRUE, PT := currentProofTime);
                ELSE
                    tonCurrentProof(IN := FALSE);
                END_IF

                IF tonCurrentProof.Q THEN
                    tonCurrentProof(IN := FALSE);
                    step := 30;
                END_IF

            30: // RUN
                deviceState := 'Running';
                running := TRUE;

                // Monitor health while running
                IF (NOT sofstarterOK) OR (NOT allInterlocksOK) THEN
                    faultActive := TRUE;
                    deviceState := 'Fault during run';
                    softstarterStart := FALSE;
                    running := FALSE;
                    step := 0;
                END_IF

                // Leave RUN when start released
                IF NOT startCommand THEN
                    softstarterStart := FALSE;
                    running := FALSE;
                    deviceState := 'Idle';
                    step := 0;
                END_IF

            ELSE
                deviceState := 'Idle';
                softstarterStart := FALSE;
                running := FALSE;
                step := 0;
        END_CASE
    END_IF

ELSE
    // No start or inhibited: safe idle
    softstarterStart := FALSE;
    running := FALSE;
    tonCurrentProof(IN := FALSE);
    IF NOT stopCommand THEN
        deviceState := 'Idle';
        step := 0;
    END_IF
END_IF

END_FUNCTION_BLOCK

// ---- Function Blocks/PaperMachine/DriveControl/FB_DryingSectionPressureControl.TcPOU
FUNCTION_BLOCK FB_DryingSectionPressureControl
VAR_INPUT
    // Curve config
    holdPressureBar           : REAL := 0.1;
    holdTimeMin               : DINT := 60;
    finalPressureBar          : REAL := 6.0;
    heatingCurveTotalTimeMin  : DINT := 360;

    // Commands & enables
    startCmd           : BOOL;
    stopCmd            : BOOL;
    resetCmd           : BOOL;
    heatingCurveEnable : BOOL;   // <-- gate for the curve

    // PID I/O & params
    steamPressureFeedback        : REAL;
    steamPressureAutoMan         : BOOL;  // FALSE=Manual, TRUE=Auto
    steamPressureAutoSetpoint    : REAL;  // Auto setpoint when curve is disabled
    steamPressureManualSetpoint  : REAL;
    steamPressureKp : REAL := 1.5;   // proportional gain
    steamPressureTn : REAL := 20.0;  // integral time [s]
    steamPressureTv : REAL := 0.2;   // derivative time [s]
	
END_VAR

VAR_OUTPUT
    steamPressureSetpointBar       : REAL; // Auto setpoint from curve (0 if stopped/disabled)
    steamPressureControllerOutput  : REAL; // PID output to solenoid
END_VAR

VAR
    // Timing
    tonMinutePulse : TON;
    minuteCounter  : DINT;
    rampElapsedMin : DINT;

    // Curve math
    pressureIncrementPerMin : REAL;

    // State
    isRunning : BOOL;
    isReset   : BOOL;

    // Filtering
    instPT1_SteamPressureFiltered : FT_PT1;
    filteredSteamPressureFeedback : REAL;
instCTRL_PID_TemperatureController : CTRL_PID;
    // PID setpoint selection
    effectiveSetpoint : REAL;
END_VAR


//────────────────────────────────────
// RESET LOGIC
//────────────────────────────────────
IF resetCmd THEN
    minuteCounter := 0;
    isRunning := FALSE;
    isReset := TRUE;
END_IF

// If curve is disabled at any time, force not running
IF NOT heatingCurveEnable THEN
    isRunning := FALSE;
END_IF

//────────────────────────────────────
// START/STOP LOGIC
//────────────────────────────────────
IF heatingCurveEnable AND startCmd AND NOT isReset THEN
    isRunning := TRUE;     // start curve
    isReset := FALSE;
END_IF

IF stopCmd THEN
    isRunning := FALSE;    // stop curve (counter preserved to resume later)
END_IF

//────────────────────────────────────
// TON MINUTE TIMER (1-minute base)
//────────────────────────────────────
IF isRunning THEN
    tonMinutePulse(IN := TRUE, PT := T#1S);

    IF tonMinutePulse.Q THEN
        minuteCounter := minuteCounter + 1;
        tonMinutePulse(IN := FALSE); // Reset TON
    END_IF;
ELSE
    tonMinutePulse(IN := FALSE);
END_IF

//────────────────────────────────────
// HEATING CURVE SETPOINT CALCULATION
// (Only when curve is enabled; otherwise keep it at 0)
//────────────────────────────────────
IF heatingCurveEnable AND isRunning THEN
    pressureIncrementPerMin := (finalPressureBar - holdPressureBar) / heatingCurveTotalTimeMin;

    IF minuteCounter <= holdTimeMin THEN
        // Phase 1: Hold
        steamPressureSetpointBar := holdPressureBar;

    ELSIF minuteCounter <= (holdTimeMin + heatingCurveTotalTimeMin) THEN
        // Phase 2: Ramp
        rampElapsedMin := minuteCounter - holdTimeMin;
        steamPressureSetpointBar := holdPressureBar + rampElapsedMin * pressureIncrementPerMin;

    ELSE
        // Phase 3: Final hold
        steamPressureSetpointBar := finalPressureBar;
    END_IF;
ELSE
    // Curve disabled or stopped => do not provide curve setpoint
    steamPressureSetpointBar := 0.0;
END_IF

//────────────────────────────────────
// PT1 FILTER — Smooth feedback input
//────────────────────────────────────
instPT1_SteamPressureFiltered(
    in  := steamPressureFeedback,
    T   := T#2S,
    K   := 1.0,
    out => filteredSteamPressureFeedback
);

//────────────────────────────────────
// PID SETPOINT SELECTION
//  - Manual: use steamPressureManualSetpoint
//  - Auto:
//      * If heatingCurveEnable = TRUE and (curve running or has progressed), use curve setpoint
//      * Else use steamPressureAutoSetpoint (external auto setpoint)
//────────────────────────────────────
IF NOT steamPressureAutoMan THEN
    // Manual mode
    effectiveSetpoint := steamPressureManualSetpoint;
ELSE
    // Auto mode
    IF heatingCurveEnable AND (isRunning OR (minuteCounter > 0)) THEN
        effectiveSetpoint := steamPressureSetpointBar;     // use the curve
    ELSE
        effectiveSetpoint := steamPressureAutoSetpoint;    // curve disabled → external auto SP
    END_IF
END_IF

//────────────────────────────────────
// PID CONTROLLER
//────────────────────────────────────
instCTRL_PID_TemperatureController(
    ACT := filteredSteamPressureFeedback,
    SET := effectiveSetpoint,
    MAN := NOT steamPressureAutoMan,
    M_I := steamPressureManualSetpoint,
    RST := FALSE,
    KP  := steamPressureKp,
    TN  := steamPressureTn,
    TV  := steamPressureTv,
    LL  := 0.0,
    LH  := 5.0,
    Y   => steamPressureControllerOutput
);

END_FUNCTION_BLOCK

// ---- Function Blocks/PaperMachine/DriveControl/FB_PressSectionDriveControl_V1.TcPOU
FUNCTION_BLOCK FB_PressSectionDriveControl_V1

(*VAR_INPUT
    {region "GROUP / INTERLOCKS"}
    //==============================================================
    // GROUP / INTERLOCKS
    //==============================================================
    startGroup                      : BOOL;  // Start command (pulse / rising edge)
    stopGroup                       : BOOL;  // Stop command (level / maintained)
    groupReset                      : BOOL;  // Group fault reset (acknowledge)
    {endregion}

    {region "DRIVE STATUS INPUTS (VFDs) — PRESS SECTION (2 MOTORS)"}
    //==============================================================
    // DRIVE STATUS INPUTS (VFDs) — PRESS SECTION (2 MOTORS)
    //==============================================================
    firstPressReady                 : BOOL;  // First press (MASTER) ready. TRUE = ready
    firstPressVfdRunFeedback        : BOOL;  // First press RUN feedback. TRUE = running
    firstPressVfdFaultFeedback      : BOOL;  // First press fault/alarm. TRUE = fault

    secondPressVfdReady             : BOOL;  // Second press (SLAVE) ready. TRUE = ready
    secondPressVfdRunFeedback       : BOOL;  // Second press RUN feedback. TRUE = running
    secondPressVfdFaultFeedback     : BOOL;  // Second press fault/alarm. TRUE = fault
    {endregion}

    {region "SPEED SETPOINTS / MODE"}
    //==============================================================
    // SPEED SETPOINTS / MODE
    //==============================================================
    groupAutoSpeedMPM               : REAL;          // Auto speed setpoint [m/min]
    groupManualSpeedMPM             : REAL := 50.0;  // Manual speed [m/min]
    groupMaxSpeed                   : REAL := 600.0; // Max allowed line speed [m/min]
    groupSpeedAutoMan               : BOOL;          // 0 = Manual, 1 = Auto
    {endregion}

    {region "FEEDBACKS (FROM DRIVES/SENSORS)"}
    //==============================================================
    // FEEDBACKS (FROM DRIVES/SENSORS)
    //==============================================================
    firstPressSpeedFeedback         : REAL;  // First press speed feedback [m/min or %]
    firstPressTorqueFeedback        : REAL;  // First press torque feedback [% or Nm]
    secondPressSpeedFeedback        : REAL;  // Second press speed feedback [m/min or %]
    secondPressTorqueFeedback       : REAL;  // Second press torque feedback [% or Nm]
    {endregion}

    {region "RATIO / OFFSETS (FOLLOWING / TRIM LOGIC)"}
    //==============================================================
    // RATIO / OFFSETS (FOLLOWING / TRIM LOGIC)
    //==============================================================
    masterSlaveGearRatio            : REAL := 1.0;   // Slave/Master speed ratio (dimensionless)
    interGroupGearRatio             : REAL := 1.0;   // Speed difference between groups

    slaveTorqueOfsset               : REAL := 0.0;   // Torque trim offset applied to slave [% or Nm]
    slaveSpeedOffset                : REAL := 0.0;   // Speed offset slave vs master [% of master]

    // Group-wide recover bump
    groupRecoverSpeedCmd            : BOOL;          // Temporarily recover speed (while TRUE)
    groupRecoverIncrement           : REAL := 5.0;   // Recovery speed increment [m/min]

    // Operator-tuned group speed offset vs previous section (TUNE2)
    grouSpeedDifCmdInc              : BOOL;          // Increment group speed offset
    grouSpeedDifCmdDec              : BOOL;          // Decrement group speed offset
    grouSpeedDifLimHigh             : REAL := 20.0;  // Upper limit for group speed offset [%]
    grouSpeedDifLimLow              : REAL := -20.0; // Lower limit for group speed offset [%]
    {endregion}

    {region "TORQUE CONTROL / LIMITS (SLAVE-FOCUSED)"}
    //==============================================================
    // TORQUE CONTROL / LIMITS (SLAVE-FOCUSED)
    //==============================================================
    enableTorquePid                 : BOOL := FALSE; // Enable torque trim PID for slave
    torqueTrimLimit                 : REAL := 10.0;  // Limit for torque trim magnitude [% or Nm]
    torqueLimitMinPct               : REAL := 0.0;   // Minimum torque limit for slave [%]
    torqueLimitMaxPct               : REAL := 150.0; // Maximum torque limit for slave [%]
    torqueFilterTime                : TIME := T#5MS; // Control torque PT1 filter time constant
    displayFilterTime               : TIME := T#20MS;// HMI display filters time constant

    //----- OSCAT CTRL_PID parameters (torque trim) -----
    torqueCtrlKp                    : REAL := 1.0;   // Proportional gain
    torqueCtrlTn                    : REAL := 8.0;   // Integral time [s]
    torqueCtrlTv                    : REAL := 0.0;   // Derivative time [s]
    {endregion}

    {region "DYNAMICS / LIMITS"}
    //==============================================================
    // DYNAMICS / LIMITS
    //==============================================================
    rampRate                        : REAL := 0.01;  // Reference acceleration rate for ramp block [%/s]
    speedDiferenceLimit             : REAL := 5.0;   // Max allowed master↔slave speed difference [%]
    {endregion}

    {region "AUX MOTORS — COMMANDS / LIMIT SWITCHES"}
    //==============================================================
    // AUX MOTORS
    //  - Direct start style with FWD/REV and end limit switches
    //==============================================================
    grouSpeedDifInc                 : BOOL;          // Increment group speed offset indication lamp
    grouSpeedDifDec                 : BOOL;          // Decrement group speed offset indication lamp

    // Felt stretcher — UPPER
    upperFelt1StretcherCmdFwd        : BOOL; // Run forward command
    upperFelt1StretcherCmdRev        : BOOL; // Run reverse command
    upperFelt1StretcherFault         : BOOL; // Reverse motion fault
    upperFelt1StretcherLimitFwd      : BOOL; // Forward end limit switch
    upperFelt1StretcherLimitRev      : BOOL; // Reverse end limit switch

    // Felt stretcher — UPPER
    upperFelt2StretcherCmdFwd        : BOOL; // Run forward command
    upperFeltt2tretcherCmdRev        : BOOL; // Run reverse command
    upperFeltS2tretcherFault         : BOOL; // Reverse motion fault
    upperFeltS2tretcherLimitFwd      : BOOL; // Forward end limit switch
    upperFeltS2tretcherLimitRev      : BOOL; // Reverse end limit switch		 

    // Felt stretcher — LOWER (direct start given; no reverse cmd provided)
    lowerFeltStretcherCmdFwd        : BOOL; // Run forward command
    lowerFeltStretcherCmdRev        : BOOL; // Run forward command
    lowerFeltStretcherFault         : BOOL; // Fault/alarm
    lowerFeltStretcherLimitFwd      : BOOL; // Forward end limit switch
    lowerFeltStretcherLimitRev      : BOOL; // Reverse end limit switch

    // Infeed roll — UPPER
    upperInfeedRollCmdFwd           : BOOL; // Run forward command
    upperInfeedRollCmdRev           : BOOL; // Run reverse command
    upperInfeedRollFault            : BOOL; // Fault/alarm
    upperInfeedRollLimitFwd         : BOOL; // Forward end limit switch
    upperInfeedRollLimitRev         : BOOL; // Reverse end limit switch

    // Infeed roll — LOWER
    lowerInfeedRollCmdFwd           : BOOL; // Run forward command
    lowerInfeedRollCmdRev           : BOOL; // Run reverse command
    lowerInfeedRollFault            : BOOL; // Fault/alarm
    lowerInfeedRollLimitFwd         : BOOL; // Forward end limit switch
    lowerInfeedRollLimitRev         : BOOL; // Reverse end limit switch
    {endregion}
		 
